LIN {X 0,Y 566.213,Z 135.454,A -85,B 0,C 180,E1 -2637.339,E2 -2637.339} C_VEL
LIN {X 0,Y 566.202,Z 135.458,A -85,B 0,C 180,E1 -2639.768,E2 -2639.768} C_VEL
LIN {X 0,Y 566.206,Z 135.453,A -85,B 0,C 180,E1 -2642.43,E2 -2642.43} C_VEL
LIN {X 0,Y 566.181,Z 135.454,A -85,B 0,C 180,E1 -2644.989,E2 -2644.989} C_VEL
LIN {X 0,Y 566.197,Z 135.457,A -85,B 0,C 180,E1 -2647.46,E2 -2647.46} C_VEL
LIN {X 0,Y 566.21,Z 135.449,A -85,B 0,C 180,E1 -2650.198,E2 -2650.198} C_VEL
LIN {X 0,Y 566.2,Z 135.453,A -85,B 0,C 180,E1 -2653.054,E2 -2653.054} C_VEL
LIN {X 0,Y 566.198,Z 135.454,A -85,B 0,C 180,E1 -2656.048,E2 -2656.048} C_VEL
LIN {X 0,Y 566.203,Z 135.457,A -85,B 0,C 180,E1 -2659.214,E2 -2659.214} C_VEL
LIN {X 0,Y 566.184,Z 135.459,A -85,B 0,C 180,E1 -2661.636,E2 -2661.636} C_VEL
LIN {X 0,Y 566.164,Z 135.455,A -85,B 0,C 180,E1 -2664.308,E2 -2664.308} C_VEL
LIN {X 0,Y 566.228,Z 135.449,A -85,B 0,C 180,E1 -2666.898,E2 -2666.898} C_VEL
LIN {X 0,Y 566.186,Z 135.459,A -85,B 0,C 180,E1 -2669.407,E2 -2669.407} C_VEL
LIN {X 0,Y 566.209,Z 135.448,A -85,B 0,C 180,E1 -2671.857,E2 -2671.857} C_VEL
LIN {X 0,Y 566.213,Z 135.447,A -85,B 0,C 180,E1 -2674.251,E2 -2674.251} C_VEL
LIN {X 0,Y 566.171,Z 135.46,A -85,B 0,C 180,E1 -2676.718,E2 -2676.718} C_VEL
LIN {X 0,Y 566.21,Z 135.448,A -85,B 0,C 180,E1 -2679.662,E2 -2679.662} C_VEL
LIN {X 0,Y 566.2,Z 135.454,A -85,B 0,C 180,E1 -2682.668,E2 -2682.668} C_VEL
LIN {X 0,Y 566.231,Z 135.447,A -85,B 0,C 180,E1 -2685.626,E2 -2685.626} C_VEL
LIN {X 0,Y 566.231,Z 135.453,A -85,B 0,C 180,E1 -2688.675,E2 -2688.675} C_VEL
LIN {X 0,Y 566.225,Z 135.445,A -85,B 0,C 180,E1 -2691.434,E2 -2691.434} C_VEL
LIN {X 0,Y 566.256,Z 135.45,A -85,B 0,C 180,E1 -2694.301,E2 -2694.301} C_VEL
LIN {X 0,Y 566.277,Z 135.442,A -85,B 0,C 180,E1 -2697.866,E2 -2697.866} C_VEL
LIN {X 0,Y 566.299,Z 135.44,A -85,B 0,C 180,E1 -2700.711,E2 -2700.711} C_VEL
LIN {X 0,Y 566.268,Z 135.444,A -85,B 0,C 180,E1 -2702.845,E2 -2702.845} C_VEL
LIN {X 0,Y 566.257,Z 135.446,A -85,B 0,C 180,E1 -2705.698,E2 -2705.698} C_VEL
LIN {X 0,Y 566.225,Z 135.448,A -85,B 0,C 180,E1 -2708.565,E2 -2708.565} C_VEL
LIN {X 0,Y 566.237,Z 135.445,A -85,B 0,C 180,E1 -2711.454,E2 -2711.454} C_VEL
LIN {X 0,Y 566.23,Z 135.45,A -85,B 0,C 180,E1 -2714.507,E2 -2714.507} C_VEL
LIN {X 0,Y 566.199,Z 135.452,A -85,B 0,C 180,E1 -2717.331,E2 -2717.331} C_VEL
LIN {X 0,Y 566.208,Z 135.451,A -85,B 0,C 180,E1 -2720.337,E2 -2720.337} C_VEL
LIN {X 0,Y 566.185,Z 135.457,A -85,B 0,C 180,E1 -2723.404,E2 -2723.404} C_VEL
LIN {X 0,Y 566.221,Z 135.455,A -85,B 0,C 180,E1 -2725.748,E2 -2725.748} C_VEL
LIN {X 0,Y 566.213,Z 135.45,A -85,B 0,C 180,E1 -2727.477,E2 -2727.477} C_VEL
LIN {X 0,Y 565.532,Z 135.536,A -85,B 0,C 180,E1 -2728.071,E2 -2728.071} C_VEL
LIN {X 0,Y 562.662,Z 135.892,A -85,B 0,C 180,E1 -2729.034,E2 -2729.034} C_VEL
LIN {X 0,Y 560.248,Z 136.199,A -85,B 0,C 180,E1 -2729.809,E2 -2729.809} C_VEL
LIN {X 0,Y 559.219,Z 136.322,A -85,B 0,C 180,E1 -2730.408,E2 -2730.408} C_VEL
LIN {X 0,Y 559.14,Z 136.331,A -85,B 0,C 180,E1 -2730.611,E2 -2730.611} C_VEL
LIN {X 0,Y 559.173,Z 136.331,A -85,B 0,C 180,E1 -2733.574,E2 -2733.574} C_VEL
LIN {X 0,Y 559.164,Z 136.328,A -85,B 0,C 180,E1 -2736.448,E2 -2736.448} C_VEL
LIN {X 0,Y 559.172,Z 136.33,A -85,B 0,C 180,E1 -2738.934,E2 -2738.934} C_VEL
LIN {X 0,Y 559.188,Z 136.327,A -85,B 0,C 180,E1 -2741.767,E2 -2741.767} C_VEL
LIN {X 0,Y 559.135,Z 136.334,A -85,B 0,C 180,E1 -2744.739,E2 -2744.739} C_VEL
LIN {X 0,Y 559.169,Z 136.319,A -85,B 0,C 180,E1 -2747.863,E2 -2747.863} C_VEL
LIN {X 0,Y 559.181,Z 136.324,A -85,B 0,C 180,E1 -2750.135,E2 -2750.135} C_VEL
LIN {X 0,Y 559.144,Z 136.339,A -85,B 0,C 180,E1 -2752.892,E2 -2752.892} C_VEL
LIN {X 0,Y 559.151,Z 136.327,A -85,B 0,C 180,E1 -2755.556,E2 -2755.556} C_VEL
LIN {X 0,Y 559.167,Z 136.329,A -85,B 0,C 180,E1 -2758.138,E2 -2758.138} C_VEL
LIN {X 0,Y 559.154,Z 136.334,A -85,B 0,C 180,E1 -2760.647,E2 -2760.647} C_VEL
LIN {X 0,Y 559.167,Z 136.331,A -85,B 0,C 180,E1 -2763.172,E2 -2763.172} C_VEL
LIN {X 0,Y 559.153,Z 136.33,A -85,B 0,C 180,E1 -2765.495,E2 -2765.495} C_VEL
LIN {X 0,Y 559.168,Z 136.337,A -85,B 0,C 180,E1 -2768.624,E2 -2768.624} C_VEL
LIN {X 0,Y 559.165,Z 136.332,A -85,B 0,C 180,E1 -2770.926,E2 -2770.926} C_VEL
LIN {X 0,Y 559.164,Z 136.332,A -85,B 0,C 180,E1 -2773.948,E2 -2773.948} C_VEL
LIN {X 0,Y 559.169,Z 136.335,A -85,B 0,C 180,E1 -2776.184,E2 -2776.184} C_VEL
LIN {X 0,Y 559.193,Z 136.326,A -85,B 0,C 180,E1 -2779.134,E2 -2779.134} C_VEL
LIN {X 0,Y 559.203,Z 136.332,A -85,B 0,C 180,E1 -2782.054,E2 -2782.054} C_VEL
LIN {X 0,Y 559.251,Z 136.319,A -85,B 0,C 180,E1 -2784.953,E2 -2784.953} C_VEL
LIN {X 0,Y 559.254,Z 136.324,A -85,B 0,C 180,E1 -2787.839,E2 -2787.839} C_VEL
LIN {X 0,Y 559.27,Z 136.317,A -85,B 0,C 180,E1 -2790.72,E2 -2790.72} C_VEL
LIN {X 0,Y 559.236,Z 136.32,A -85,B 0,C 180,E1 -2792.881,E2 -2792.881} C_VEL
LIN {X 0,Y 559.229,Z 136.329,A -85,B 0,C 180,E1 -2795.77,E2 -2795.77} C_VEL
LIN {X 0,Y 559.189,Z 136.326,A -85,B 0,C 180,E1 -2798.674,E2 -2798.674} C_VEL
LIN {X 0,Y 559.202,Z 136.332,A -85,B 0,C 180,E1 -2801.6,E2 -2801.6} C_VEL
LIN {X 0,Y 559.196,Z 136.325,A -85,B 0,C 180,E1 -2804.595,E2 -2804.595} C_VEL
LIN {X 0,Y 559.156,Z 136.338,A -85,B 0,C 180,E1 -2807.557,E2 -2807.557} C_VEL
LIN {X 0,Y 559.169,Z 136.332,A -85,B 0,C 180,E1 -2809.837,E2 -2809.837} C_VEL
LIN {X 0,Y 559.139,Z 136.333,A -85,B 0,C 180,E1 -2812.153,E2 -2812.153} C_VEL
LIN {X 0,Y 559.175,Z 136.334,A -85,B 0,C 180,E1 -2815.187,E2 -2815.187} C_VEL
LIN {X 0,Y 559.188,Z 136.328,A -85,B 0,C 180,E1 -2817.711,E2 -2817.711} C_VEL
LIN {X 0,Y 559.165,Z 136.327,A -85,B 0,C 180,E1 -2820.182,E2 -2820.182} C_VEL
LIN {X 0,Y 559.171,Z 136.331,A -85,B 0,C 180,E1 -2822.714,E2 -2822.714} C_VEL
LIN {X 0,Y 559.14,Z 136.335,A -85,B 0,C 180,E1 -2825.323,E2 -2825.323} C_VEL
LIN {X 0,Y 559.132,Z 136.332,A -85,B 0,C 180,E1 -2828.017,E2 -2828.017} C_VEL
LIN {X 0,Y 559.171,Z 136.331,A -85,B 0,C 180,E1 -2830.811,E2 -2830.811} C_VEL
LIN {X 0,Y 559.136,Z 136.328,A -85,B 0,C 180,E1 -2833.734,E2 -2833.734} C_VEL
LIN {X 0,Y 559.167,Z 136.337,A -85,B 0,C 180,E1 -2836.801,E2 -2836.801} C_VEL
LIN {X 0,Y 559.172,Z 136.327,A -85,B 0,C 180,E1 -2839.19,E2 -2839.19} C_VEL
LIN {X 0,Y 559.129,Z 136.334,A -85,B 0,C 180,E1 -2841.983,E2 -2841.983} C_VEL
LIN {X 0,Y 559.154,Z 136.331,A -85,B 0,C 180,E1 -2844.783,E2 -2844.783} C_VEL
LIN {X 0,Y 559.169,Z 136.327,A -85,B 0,C 180,E1 -2847.361,E2 -2847.361} C_VEL
LIN {X 0,Y 559.145,Z 136.336,A -85,B 0,C 180,E1 -2850.142,E2 -2850.142} C_VEL
LIN {X 0,Y 559.178,Z 136.323,A -85,B 0,C 180,E1 -2853.17,E2 -2853.17} C_VEL
LIN {X 0,Y 559.152,Z 136.329,A -85,B 0,C 180,E1 -2855.495,E2 -2855.495} C_VEL
LIN {X 0,Y 559.166,Z 136.329,A -85,B 0,C 180,E1 -2858.624,E2 -2858.624} C_VEL
LIN {X 0,Y 559.166,Z 136.322,A -85,B 0,C 180,E1 -2860.927,E2 -2860.927} C_VEL
LIN {X 0,Y 559.164,Z 136.335,A -85,B 0,C 180,E1 -2863.948,E2 -2863.948} C_VEL
LIN {X 0,Y 559.169,Z 136.333,A -85,B 0,C 180,E1 -2866.184,E2 -2866.184} C_VEL
LIN {X 0,Y 559.19,Z 136.321,A -85,B 0,C 180,E1 -2869.134,E2 -2869.134} C_VEL
LIN {X 0,Y 559.2,Z 136.328,A -85,B 0,C 180,E1 -2872.054,E2 -2872.054} C_VEL
LIN {X 0,Y 559.25,Z 136.318,A -85,B 0,C 180,E1 -2874.954,E2 -2874.954} C_VEL
LIN {X 0,Y 559.247,Z 136.321,A -85,B 0,C 180,E1 -2877.84,E2 -2877.84} C_VEL
LIN {X 0,Y 559.269,Z 136.31,A -85,B 0,C 180,E1 -2880.72,E2 -2880.72} C_VEL
LIN {X 0,Y 559.237,Z 136.319,A -85,B 0,C 180,E1 -2882.882,E2 -2882.882} C_VEL
LIN {X 0,Y 559.225,Z 136.324,A -85,B 0,C 180,E1 -2885.771,E2 -2885.771} C_VEL
LIN {X 0,Y 559.184,Z 136.322,A -85,B 0,C 180,E1 -2888.675,E2 -2888.675} C_VEL
LIN {X 0,Y 559.202,Z 136.327,A -85,B 0,C 180,E1 -2891.601,E2 -2891.601} C_VEL
LIN {X 0,Y 559.197,Z 136.325,A -85,B 0,C 180,E1 -2894.596,E2 -2894.596} C_VEL
LIN {X 0,Y 559.16,Z 136.327,A -85,B 0,C 180,E1 -2897.557,E2 -2897.557} C_VEL
LIN {X 0,Y 559.169,Z 136.325,A -85,B 0,C 180,E1 -2899.838,E2 -2899.838} C_VEL
LIN {X 0,Y 559.138,Z 136.331,A -85,B 0,C 180,E1 -2902.153,E2 -2902.153} C_VEL
LIN {X 0,Y 559.174,Z 136.328,A -85,B 0,C 180,E1 -2905.299,E2 -2905.299} C_VEL
LIN {X 0,Y 559.155,Z 136.326,A -85,B 0,C 180,E1 -2907.714,E2 -2907.714} C_VEL
LIN {X 0,Y 559.155,Z 136.33,A -85,B 0,C 180,E1 -2910.183,E2 -2910.183} C_VEL
LIN {X 0,Y 559.174,Z 136.334,A -85,B 0,C 180,E1 -2912.714,E2 -2912.714} C_VEL
LIN {X 0,Y 559.129,Z 136.333,A -85,B 0,C 180,E1 -2915.324,E2 -2915.324} C_VEL
LIN {X 0,Y 559.131,Z 136.334,A -85,B 0,C 180,E1 -2918.018,E2 -2918.018} C_VEL
LIN {X 0,Y 559.154,Z 136.334,A -85,B 0,C 180,E1 -2920.813,E2 -2920.813} C_VEL
LIN {X 0,Y 559.14,Z 136.331,A -85,B 0,C 180,E1 -2923.734,E2 -2923.734} C_VEL
LIN {X 0,Y 559.144,Z 136.334,A -85,B 0,C 180,E1 -2926.804,E2 -2926.804} C_VEL
LIN {X 0,Y 559.155,Z 136.325,A -85,B 0,C 180,E1 -2929.188,E2 -2929.188} C_VEL
LIN {X 0,Y 559.135,Z 136.337,A -85,B 0,C 180,E1 -2931.983,E2 -2931.983} C_VEL
LIN {X 0,Y 559.133,Z 136.333,A -85,B 0,C 180,E1 -2934.788,E2 -2934.788} C_VEL
LIN {X 0,Y 559.158,Z 136.329,A -85,B 0,C 180,E1 -2937.365,E2 -2937.365} C_VEL
LIN {X 0,Y 559.15,Z 136.337,A -85,B 0,C 180,E1 -2940.143,E2 -2940.143} C_VEL
LIN {X 0,Y 559.172,Z 136.331,A -85,B 0,C 180,E1 -2943.173,E2 -2943.173} C_VEL
LIN {X 0,Y 559.231,Z 136.477,A -85,B 0,C 180,E1 -2944.837,E2 -2944.837} C_VEL
LIN {X 0,Y 559.901,Z 140.893,A -85,B 0,C 180,E1 -2945.727,E2 -2945.727} C_VEL
LIN {X 0,Y 559.626,Z 156.438,A -85,B 0,C 180,E1 -2948.642,E2 -2948.642} C_VEL
LIN {X 0,Y 559.476,Z 170.036,A -85,B 0,C 180,E1 -2951.128,E2 -2951.128} C_VEL
LIN {X 0,Y 559.339,Z 184.658,A -85,B 0,C 180,E1 -2953.766,E2 -2953.766} C_VEL
LIN {X 0,Y 559.241,Z 196.165,A -85,B 0,C 180,E1 -2955.792,E2 -2955.792} C_VEL
LIN {X 0,Y 559.599,Z 198.54,A -85,B 0,C 180,E1 -2955.869,E2 -2955.869} C_VEL
LIN {X 0,Y 560.276,Z 204.023,A -85,B 0,C 180,E1 -2955.957,E2 -2955.957} C_VEL
LIN {X 0,Y 560.043,Z 301.149,A -85,B 0,C 180,E1 -2957.222,E2 -2957.222} C_VEL
LIN {X 0,Y 559.981,Z 311.04,A -85,B 0,C 180,E1 -2957.428,E2 -2957.428} C_VEL
LIN {X 0,Y 559.892,Z 321.006,A -85,B 0,C 180,E1 -2957.725,E2 -2957.725} C_VEL
LIN {X 0,Y 559.753,Z 330.356,A -85,B 0,C 180,E1 -2958.09,E2 -2958.09} C_VEL
LIN {X 0,Y 559.646,Z 339.669,A -85,B 0,C 180,E1 -2958.547,E2 -2958.547} C_VEL
LIN {X 0,Y 559.486,Z 349.449,A -85,B 0,C 180,E1 -2959.139,E2 -2959.139} C_VEL
LIN {X 0,Y 559.377,Z 358.154,A -85,B 0,C 180,E1 -2959.778,E2 -2959.778} C_VEL
LIN {X 0,Y 559.279,Z 365.525,A -85,B 0,C 180,E1 -2960.416,E2 -2960.416} C_VEL
LIN {X 0,Y 559.137,Z 372.717,A -85,B 0,C 180,E1 -2961.143,E2 -2961.143} C_VEL
LIN {X 0,Y 559.052,Z 380.264,A -85,B 0,C 180,E1 -2962.052,E2 -2962.052} C_VEL
LIN {X 0,Y 558.943,Z 386.554,A -85,B 0,C 180,E1 -2962.958,E2 -2962.958} C_VEL
LIN {X 0,Y 558.909,Z 391.787,A -85,B 0,C 180,E1 -2963.864,E2 -2963.864} C_VEL
LIN {X 0,Y 558.798,Z 396.885,A -85,B 0,C 180,E1 -2964.949,E2 -2964.949} C_VEL
LIN {X 0,Y 558.844,Z 400.843,A -85,B 0,C 180,E1 -2966.034,E2 -2966.034} C_VEL
LIN {X 0,Y 558.799,Z 403.767,A -85,B 0,C 180,E1 -2967.116,E2 -2967.116} C_VEL
LIN {X 0,Y 558.745,Z 406.194,A -85,B 0,C 180,E1 -2968.559,E2 -2968.559} C_VEL
LIN {X 0,Y 558.741,Z 406.778,A -85,B 0,C 180,E1 -2969.279,E2 -2969.279} C_VEL
LIN {X 0,Y 558.741,Z 406.778,A -85,B 0,C 180,E1 -2970.721,E2 -2970.721} C_VEL
LIN {X 0,Y 558.745,Z 406.194,A -85,B 0,C 180,E1 -2971.441,E2 -2971.441} C_VEL
LIN {X 0,Y 558.799,Z 403.767,A -85,B 0,C 180,E1 -2972.884,E2 -2972.884} C_VEL
LIN {X 0,Y 558.844,Z 400.843,A -85,B 0,C 180,E1 -2973.966,E2 -2973.966} C_VEL
LIN {X 0,Y 558.798,Z 396.885,A -85,B 0,C 180,E1 -2975.051,E2 -2975.051} C_VEL
LIN {X 0,Y 558.91,Z 391.787,A -85,B 0,C 180,E1 -2976.136,E2 -2976.136} C_VEL
LIN {X 0,Y 558.934,Z 386.668,A -85,B 0,C 180,E1 -2977.024,E2 -2977.024} C_VEL
LIN {X 0,Y 559.052,Z 380.264,A -85,B 0,C 180,E1 -2977.948,E2 -2977.948} C_VEL
LIN {X 0,Y 559.137,Z 372.717,A -85,B 0,C 180,E1 -2978.857,E2 -2978.857} C_VEL
LIN {X 0,Y 559.29,Z 363.612,A -85,B 0,C 180,E1 -2979.767,E2 -2979.767} C_VEL
LIN {X 0,Y 559.449,Z 352.147,A -85,B 0,C 180,E1 -2980.678,E2 -2980.678} C_VEL
LIN {X 0,Y 559.571,Z 343.177,A -85,B 0,C 180,E1 -2981.257,E2 -2981.257} C_VEL
LIN {X 0,Y 559.728,Z 333.771,A -85,B 0,C 180,E1 -2981.754,E2 -2981.754} C_VEL
LIN {X 0,Y 559.829,Z 323.581,A -85,B 0,C 180,E1 -2982.184,E2 -2982.184} C_VEL
LIN {X 0,Y 559.968,Z 313.661,A -85,B 0,C 180,E1 -2982.503,E2 -2982.503} C_VEL
LIN {X 0,Y 560.026,Z 303.813,A -85,B 0,C 180,E1 -2982.732,E2 -2982.732} C_VEL
LIN {X 0,Y 560.164,Z 279.204,A -85,B 0,C 180,E1 -2983.075,E2 -2983.075} C_VEL
LIN {X 0,Y 560.207,Z 202.231,A -85,B 0,C 180,E1 -2984.067,E2 -2984.067} C_VEL
LIN {X 0,Y 559.275,Z 196.499,A -85,B 0,C 180,E1 -2984.184,E2 -2984.184} C_VEL
LIN {X 0,Y 559.225,Z 195.089,A -85,B 0,C 180,E1 -2984.371,E2 -2984.371} C_VEL
LIN {X 0,Y 559.384,Z 178.831,A -85,B 0,C 180,E1 -2987.282,E2 -2987.282} C_VEL
LIN {X 0,Y 559.584,Z 162.717,A -85,B 0,C 180,E1 -2990.205,E2 -2990.205} C_VEL
LIN {X 0,Y 559.842,Z 146.337,A -85,B 0,C 180,E1 -2993.251,E2 -2993.251} C_VEL
LIN {X 0,Y 559.822,Z 139.871,A -85,B 0,C 180,E1 -2994.474,E2 -2994.474} C_VEL
LIN {X 0,Y 559.213,Z 136.373,A -85,B 0,C 180,E1 -2995.193,E2 -2995.193} C_VEL
LIN {X 0,Y 559.183,Z 136.333,A -85,B 0,C 180,E1 -2997.712,E2 -2997.712} C_VEL
LIN {X 0,Y 559.157,Z 136.337,A -85,B 0,C 180,E1 -3000.182,E2 -3000.182} C_VEL
LIN {X 0,Y 559.158,Z 136.329,A -85,B 0,C 180,E1 -3002.715,E2 -3002.715} C_VEL
LIN {X 0,Y 559.128,Z 136.334,A -85,B 0,C 180,E1 -3005.324,E2 -3005.324} C_VEL
LIN {X 0,Y 559.135,Z 136.337,A -85,B 0,C 180,E1 -3008.017,E2 -3008.017} C_VEL
LIN {X 0,Y 559.155,Z 136.325,A -85,B 0,C 180,E1 -3010.812,E2 -3010.812} C_VEL
LIN {X 0,Y 559.138,Z 136.338,A -85,B 0,C 180,E1 -3013.734,E2 -3013.734} C_VEL
LIN {X 0,Y 559.146,Z 136.331,A -85,B 0,C 180,E1 -3016.803,E2 -3016.803} C_VEL
LIN {X 0,Y 559.154,Z 136.334,A -85,B 0,C 180,E1 -3019.187,E2 -3019.187} C_VEL
LIN {X 0,Y 559.131,Z 136.334,A -85,B 0,C 180,E1 -3021.982,E2 -3021.982} C_VEL
LIN {X 0,Y 559.133,Z 136.333,A -85,B 0,C 180,E1 -3024.786,E2 -3024.786} C_VEL
LIN {X 0,Y 559.173,Z 136.334,A -85,B 0,C 180,E1 -3027.361,E2 -3027.361} C_VEL
LIN {X 0,Y 559.148,Z 136.33,A -85,B 0,C 180,E1 -3030.142,E2 -3030.142} C_VEL
LIN {X 0,Y 559.168,Z 136.332,A -85,B 0,C 180,E1 -3033.097,E2 -3033.097} C_VEL
LIN {X 0,Y 559.155,Z 136.331,A -85,B 0,C 180,E1 -3035.494,E2 -3035.494} C_VEL
LIN {X 0,Y 559.169,Z 136.331,A -85,B 0,C 180,E1 -3038.623,E2 -3038.623} C_VEL
LIN {X 0,Y 559.166,Z 136.331,A -85,B 0,C 180,E1 -3040.926,E2 -3040.926} C_VEL
LIN {X 0,Y 559.164,Z 136.327,A -85,B 0,C 180,E1 -3043.947,E2 -3043.947} C_VEL
LIN {X 0,Y 559.171,Z 136.328,A -85,B 0,C 180,E1 -3046.184,E2 -3046.184} C_VEL
LIN {X 0,Y 559.191,Z 136.322,A -85,B 0,C 180,E1 -3049.133,E2 -3049.133} C_VEL
LIN {X 0,Y 559.2,Z 136.322,A -85,B 0,C 180,E1 -3052.053,E2 -3052.053} C_VEL
LIN {X 0,Y 559.25,Z 136.32,A -85,B 0,C 180,E1 -3054.953,E2 -3054.953} C_VEL
LIN {X 0,Y 559.248,Z 136.318,A -85,B 0,C 180,E1 -3057.839,E2 -3057.839} C_VEL
LIN {X 0,Y 559.269,Z 136.315,A -85,B 0,C 180,E1 -3060.72,E2 -3060.72} C_VEL
LIN {X 0,Y 559.235,Z 136.32,A -85,B 0,C 180,E1 -3062.881,E2 -3062.881} C_VEL
LIN {X 0,Y 559.225,Z 136.323,A -85,B 0,C 180,E1 -3065.77,E2 -3065.77} C_VEL
LIN {X 0,Y 559.184,Z 136.323,A -85,B 0,C 180,E1 -3068.674,E2 -3068.674} C_VEL
LIN {X 0,Y 559.201,Z 136.322,A -85,B 0,C 180,E1 -3071.6,E2 -3071.6} C_VEL
LIN {X 0,Y 559.195,Z 136.326,A -85,B 0,C 180,E1 -3074.595,E2 -3074.595} C_VEL
LIN {X 0,Y 559.159,Z 136.331,A -85,B 0,C 180,E1 -3077.556,E2 -3077.556} C_VEL
LIN {X 0,Y 559.167,Z 136.331,A -85,B 0,C 180,E1 -3079.837,E2 -3079.837} C_VEL
LIN {X 0,Y 559.137,Z 136.335,A -85,B 0,C 180,E1 -3082.153,E2 -3082.153} C_VEL
LIN {X 0,Y 559.175,Z 136.328,A -85,B 0,C 180,E1 -3085.187,E2 -3085.187} C_VEL
LIN {X 0,Y 559.19,Z 136.33,A -85,B 0,C 180,E1 -3087.711,E2 -3087.711} C_VEL
LIN {X 0,Y 559.14,Z 136.331,A -85,B 0,C 180,E1 -3090.611,E2 -3090.611} C_VEL
LIN {X 0,Y 558.481,Z 136.419,A -85,B 0,C 180,E1 -3091.212,E2 -3091.212} C_VEL
LIN {X 0,Y 555.622,Z 136.771,A -85,B 0,C 180,E1 -3092.188,E2 -3092.188} C_VEL
LIN {X 0,Y 553.211,Z 137.071,A -85,B 0,C 180,E1 -3092.974,E2 -3092.974} C_VEL
LIN {X 0,Y 552.192,Z 137.2,A -85,B 0,C 180,E1 -3093.581,E2 -3093.581} C_VEL
LIN {X 0,Y 552.118,Z 137.203,A -85,B 0,C 180,E1 -3093.786,E2 -3093.786} C_VEL
LIN {X 0,Y 552.107,Z 137.208,A -85,B 0,C 180,E1 -3096.746,E2 -3096.746} C_VEL
LIN {X 0,Y 552.129,Z 137.208,A -85,B 0,C 180,E1 -3099.527,E2 -3099.527} C_VEL
LIN {X 0,Y 552.126,Z 137.205,A -85,B 0,C 180,E1 -3102.425,E2 -3102.425} C_VEL
LIN {X 0,Y 552.092,Z 137.209,A -85,B 0,C 180,E1 -3105.563,E2 -3105.563} C_VEL
LIN {X 0,Y 552.134,Z 137.198,A -85,B 0,C 180,E1 -3108.676,E2 -3108.676} C_VEL
LIN {X 0,Y 552.116,Z 137.21,A -85,B 0,C 180,E1 -3111.411,E2 -3111.411} C_VEL
LIN {X 0,Y 552.109,Z 137.205,A -85,B 0,C 180,E1 -3114.159,E2 -3114.159} C_VEL
LIN {X 0,Y 552.119,Z 137.21,A -85,B 0,C 180,E1 -3116.815,E2 -3116.815} C_VEL
LIN {X 0,Y 552.11,Z 137.207,A -85,B 0,C 180,E1 -3119.392,E2 -3119.392} C_VEL
LIN {X 0,Y 552.119,Z 137.205,A -85,B 0,C 180,E1 -3121.903,E2 -3121.903} C_VEL
LIN {X 0,Y 552.152,Z 137.211,A -85,B 0,C 180,E1 -3124.65,E2 -3124.65} C_VEL
LIN {X 0,Y 552.093,Z 137.21,A -85,B 0,C 180,E1 -3127.549,E2 -3127.549} C_VEL
LIN {X 0,Y 552.153,Z 137.209,A -85,B 0,C 180,E1 -3130.675,E2 -3130.675} C_VEL
LIN {X 0,Y 552.114,Z 137.208,A -85,B 0,C 180,E1 -3133.737,E2 -3133.737} C_VEL
LIN {X 0,Y 552.133,Z 137.209,A -85,B 0,C 180,E1 -3136.005,E2 -3136.005} C_VEL
LIN {X 0,Y 552.16,Z 137.203,A -85,B 0,C 180,E1 -3138.993,E2 -3138.993} C_VEL
LIN {X 0,Y 552.157,Z 137.208,A -85,B 0,C 180,E1 -3141.952,E2 -3141.952} C_VEL
LIN {X 0,Y 552.226,Z 137.194,A -85,B 0,C 180,E1 -3144.889,E2 -3144.889} C_VEL
LIN {X 0,Y 552.225,Z 137.2,A -85,B 0,C 180,E1 -3147.812,E2 -3147.812} C_VEL
LIN {X 0,Y 552.24,Z 137.193,A -85,B 0,C 180,E1 -3150.729,E2 -3150.729} C_VEL
LIN {X 0,Y 552.203,Z 137.197,A -85,B 0,C 180,E1 -3152.918,E2 -3152.918} C_VEL
LIN {X 0,Y 552.199,Z 137.205,A -85,B 0,C 180,E1 -3155.844,E2 -3155.844} C_VEL
LIN {X 0,Y 552.16,Z 137.202,A -85,B 0,C 180,E1 -3158.786,E2 -3158.786} C_VEL
LIN {X 0,Y 552.16,Z 137.21,A -85,B 0,C 180,E1 -3161.75,E2 -3161.75} C_VEL
LIN {X 0,Y 552.133,Z 137.205,A -85,B 0,C 180,E1 -3164.748,E2 -3164.748} C_VEL
LIN {X 0,Y 552.108,Z 137.214,A -85,B 0,C 180,E1 -3167.788,E2 -3167.788} C_VEL
LIN {X 0,Y 552.128,Z 137.207,A -85,B 0,C 180,E1 -3170.101,E2 -3170.101} C_VEL
LIN {X 0,Y 552.093,Z 137.21,A -85,B 0,C 180,E1 -3172.451,E2 -3172.451} C_VEL
LIN {X 0,Y 552.152,Z 137.211,A -85,B 0,C 180,E1 -3175.35,E2 -3175.35} C_VEL
LIN {X 0,Y 552.121,Z 137.205,A -85,B 0,C 180,E1 -3178.097,E2 -3178.097} C_VEL
LIN {X 0,Y 552.11,Z 137.207,A -85,B 0,C 180,E1 -3180.608,E2 -3180.608} C_VEL
LIN {X 0,Y 552.118,Z 137.21,A -85,B 0,C 180,E1 -3183.185,E2 -3183.185} C_VEL
LIN {X 0,Y 552.099,Z 137.207,A -85,B 0,C 180,E1 -3185.842,E2 -3185.842} C_VEL
LIN {X 0,Y 552.122,Z 137.211,A -85,B 0,C 180,E1 -3189.062,E2 -3189.062} C_VEL
LIN {X 0,Y 552.133,Z 137.196,A -85,B 0,C 180,E1 -3191.444,E2 -3191.444} C_VEL
LIN {X 0,Y 552.09,Z 137.21,A -85,B 0,C 180,E1 -3194.532,E2 -3194.532} C_VEL
LIN {X 0,Y 552.126,Z 137.204,A -85,B 0,C 180,E1 -3197.584,E2 -3197.584} C_VEL
LIN {X 0,Y 552.129,Z 137.208,A -85,B 0,C 180,E1 -3200.473,E2 -3200.473} C_VEL
LIN {X 0,Y 552.11,Z 137.207,A -85,B 0,C 180,E1 -3203.316,E2 -3203.316} C_VEL
LIN {X 0,Y 552.135,Z 137.201,A -85,B 0,C 180,E1 -3205.94,E2 -3205.94} C_VEL
LIN {X 0,Y 552.113,Z 137.215,A -85,B 0,C 180,E1 -3208.541,E2 -3208.541} C_VEL
LIN {X 0,Y 552.121,Z 137.203,A -85,B 0,C 180,E1 -3211.438,E2 -3211.438} C_VEL
LIN {X 0,Y 552.133,Z 137.211,A -85,B 0,C 180,E1 -3214.356,E2 -3214.356} C_VEL
LIN {X 0,Y 552.105,Z 137.209,A -85,B 0,C 180,E1 -3216.759,E2 -3216.759} C_VEL
LIN {X 0,Y 552.115,Z 137.204,A -85,B 0,C 180,E1 -3219.12,E2 -3219.12} C_VEL
LIN {X 0,Y 552.126,Z 137.2,A -85,B 0,C 180,E1 -3221.445,E2 -3221.445} C_VEL
LIN {X 0,Y 552.113,Z 137.209,A -85,B 0,C 180,E1 -3223.738,E2 -3223.738} C_VEL
LIN {X 0,Y 552.132,Z 137.213,A -85,B 0,C 180,E1 -3226.005,E2 -3226.005} C_VEL
LIN {X 0,Y 552.157,Z 137.197,A -85,B 0,C 180,E1 -3228.994,E2 -3228.994} C_VEL
LIN {X 0,Y 552.154,Z 137.207,A -85,B 0,C 180,E1 -3231.952,E2 -3231.952} C_VEL
LIN {X 0,Y 552.225,Z 137.192,A -85,B 0,C 180,E1 -3234.889,E2 -3234.889} C_VEL
LIN {X 0,Y 552.219,Z 137.196,A -85,B 0,C 180,E1 -3237.812,E2 -3237.812} C_VEL
LIN {X 0,Y 552.239,Z 137.185,A -85,B 0,C 180,E1 -3240.73,E2 -3240.73} C_VEL
LIN {X 0,Y 552.203,Z 137.195,A -85,B 0,C 180,E1 -3242.919,E2 -3242.919} C_VEL
LIN {X 0,Y 552.196,Z 137.199,A -85,B 0,C 180,E1 -3245.844,E2 -3245.844} C_VEL
LIN {X 0,Y 552.155,Z 137.198,A -85,B 0,C 180,E1 -3248.786,E2 -3248.786} C_VEL
LIN {X 0,Y 552.16,Z 137.202,A -85,B 0,C 180,E1 -3251.751,E2 -3251.751} C_VEL
LIN {X 0,Y 552.134,Z 137.206,A -85,B 0,C 180,E1 -3254.749,E2 -3254.749} C_VEL
LIN {X 0,Y 552.11,Z 137.202,A -85,B 0,C 180,E1 -3257.789,E2 -3257.789} C_VEL
LIN {X 0,Y 552.128,Z 137.201,A -85,B 0,C 180,E1 -3260.102,E2 -3260.102} C_VEL
LIN {X 0,Y 552.09,Z 137.21,A -85,B 0,C 180,E1 -3262.451,E2 -3262.451} C_VEL
LIN {X 0,Y 552.154,Z 137.201,A -85,B 0,C 180,E1 -3265.351,E2 -3265.351} C_VEL
LIN {X 0,Y 552.107,Z 137.204,A -85,B 0,C 180,E1 -3268.099,E2 -3268.099} C_VEL
LIN {X 0,Y 552.106,Z 137.213,A -85,B 0,C 180,E1 -3270.609,E2 -3270.609} C_VEL
LIN {X 0,Y 552.122,Z 137.205,A -85,B 0,C 180,E1 -3273.186,E2 -3273.186} C_VEL
LIN {X 0,Y 552.086,Z 137.209,A -85,B 0,C 180,E1 -3275.844,E2 -3275.844} C_VEL
LIN {X 0,Y 552.12,Z 137.206,A -85,B 0,C 180,E1 -3279.062,E2 -3279.062} C_VEL
LIN {X 0,Y 552.12,Z 137.205,A -85,B 0,C 180,E1 -3281.446,E2 -3281.446} C_VEL
LIN {X 0,Y 552.093,Z 137.216,A -85,B 0,C 180,E1 -3284.532,E2 -3284.532} C_VEL
LIN {X 0,Y 552.129,Z 137.205,A -85,B 0,C 180,E1 -3287.585,E2 -3287.585} C_VEL
LIN {X 0,Y 552.134,Z 137.21,A -85,B 0,C 180,E1 -3290.474,E2 -3290.474} C_VEL
LIN {X 0,Y 552.107,Z 137.207,A -85,B 0,C 180,E1 -3293.317,E2 -3293.317} C_VEL
LIN {X 0,Y 552.128,Z 137.21,A -85,B 0,C 180,E1 -3295.94,E2 -3295.94} C_VEL
LIN {X 0,Y 552.121,Z 137.21,A -85,B 0,C 180,E1 -3298.541,E2 -3298.541} C_VEL
LIN {X 0,Y 552.106,Z 137.211,A -85,B 0,C 180,E1 -3301.442,E2 -3301.442} C_VEL
LIN {X 0,Y 552.135,Z 137.213,A -85,B 0,C 180,E1 -3304.356,E2 -3304.356} C_VEL
LIN {X 0,Y 552.163,Z 137.377,A -85,B 0,C 180,E1 -3304.684,E2 -3304.684} C_VEL
LIN {X 0,Y 552.952,Z 142.881,A -85,B 0,C 180,E1 -3305.802,E2 -3305.802} C_VEL
LIN {X 0,Y 552.651,Z 160.492,A -85,B 0,C 180,E1 -3309.141,E2 -3309.141} C_VEL
LIN {X 0,Y 552.461,Z 176.175,A -85,B 0,C 180,E1 -3312.032,E2 -3312.032} C_VEL
LIN {X 0,Y 552.221,Z 193.889,A -85,B 0,C 180,E1 -3315.254,E2 -3315.254} C_VEL
LIN {X 0,Y 552.194,Z 196.156,A -85,B 0,C 180,E1 -3315.621,E2 -3315.621} C_VEL
LIN {X 0,Y 553.383,Z 204.134,A -85,B 0,C 180,E1 -3315.783,E2 -3315.783} C_VEL
LIN {X 0,Y 553.136,Z 300.958,A -85,B 0,C 180,E1 -3317.06,E2 -3317.06} C_VEL
LIN {X 0,Y 553.044,Z 310.855,A -85,B 0,C 180,E1 -3317.268,E2 -3317.268} C_VEL
LIN {X 0,Y 552.962,Z 320.834,A -85,B 0,C 180,E1 -3317.569,E2 -3317.569} C_VEL
LIN {X 0,Y 552.765,Z 331.199,A -85,B 0,C 180,E1 -3317.983,E2 -3317.983} C_VEL
LIN {X 0,Y 552.64,Z 340.439,A -85,B 0,C 180,E1 -3318.452,E2 -3318.452} C_VEL
LIN {X 0,Y 552.496,Z 349.338,A -85,B 0,C 180,E1 -3319,E2 -3319} C_VEL
LIN {X 0,Y 552.383,Z 358.071,A -85,B 0,C 180,E1 -3319.647,E2 -3319.647} C_VEL
LIN {X 0,Y 552.243,Z 365.468,A -85,B 0,C 180,E1 -3320.292,E2 -3320.292} C_VEL
LIN {X 0,Y 552.099,Z 372.688,A -85,B 0,C 180,E1 -3321.029,E2 -3321.029} C_VEL
LIN {X 0,Y 552.01,Z 378.884,A -85,B 0,C 180,E1 -3321.765,E2 -3321.765} C_VEL
LIN {X 0,Y 551.904,Z 385.392,A -85,B 0,C 180,E1 -3322.684,E2 -3322.684} C_VEL
LIN {X 0,Y 551.808,Z 391.081,A -85,B 0,C 180,E1 -3323.651,E2 -3323.651} C_VEL
LIN {X 0,Y 551.802,Z 395.331,A -85,B 0,C 180,E1 -3324.519,E2 -3324.519} C_VEL
LIN {X 0,Y 551.766,Z 399.626,A -85,B 0,C 180,E1 -3325.617,E2 -3325.617} C_VEL
LIN {X 0,Y 551.75,Z 401.973,A -85,B 0,C 180,E1 -3326.349,E2 -3326.349} C_VEL
LIN {X 0,Y 551.723,Z 403.76,A -85,B 0,C 180,E1 -3327.079,E2 -3327.079} C_VEL
LIN {X 0,Y 551.645,Z 406.185,A -85,B 0,C 180,E1 -3328.54,E2 -3328.54} C_VEL
LIN {X 0,Y 551.641,Z 406.769,A -85,B 0,C 180,E1 -3329.27,E2 -3329.27} C_VEL
LIN {X 0,Y 551.641,Z 406.769,A -85,B 0,C 180,E1 -3330.73,E2 -3330.73} C_VEL
LIN {X 0,Y 551.645,Z 406.185,A -85,B 0,C 180,E1 -3331.46,E2 -3331.46} C_VEL
LIN {X 0,Y 551.723,Z 403.76,A -85,B 0,C 180,E1 -3332.921,E2 -3332.921} C_VEL
LIN {X 0,Y 551.764,Z 400.835,A -85,B 0,C 180,E1 -3334.017,E2 -3334.017} C_VEL
LIN {X 0,Y 551.723,Z 396.875,A -85,B 0,C 180,E1 -3335.116,E2 -3335.116} C_VEL
LIN {X 0,Y 551.837,Z 392.381,A -85,B 0,C 180,E1 -3336.098,E2 -3336.098} C_VEL
LIN {X 0,Y 551.886,Z 386.542,A -85,B 0,C 180,E1 -3337.132,E2 -3337.132} C_VEL
LIN {X 0,Y 551.984,Z 380.254,A -85,B 0,C 180,E1 -3338.051,E2 -3338.051} C_VEL
LIN {X 0,Y 552.071,Z 374.315,A -85,B 0,C 180,E1 -3338.787,E2 -3338.787} C_VEL
LIN {X 0,Y 552.199,Z 367.387,A -85,B 0,C 180,E1 -3339.524,E2 -3339.524} C_VEL
LIN {X 0,Y 552.339,Z 359.205,A -85,B 0,C 180,E1 -3340.261,E2 -3340.261} C_VEL
LIN {X 0,Y 552.462,Z 350.69,A -85,B 0,C 180,E1 -3340.908,E2 -3340.908} C_VEL
LIN {X 0,Y 552.621,Z 341.516,A -85,B 0,C 180,E1 -3341.487,E2 -3341.487} C_VEL
LIN {X 0,Y 552.789,Z 332.208,A -85,B 0,C 180,E1 -3341.969,E2 -3341.969} C_VEL
LIN {X 0,Y 552.88,Z 323.409,A -85,B 0,C 180,E1 -3342.34,E2 -3342.34} C_VEL
LIN {X 0,Y 553.031,Z 313.479,A -85,B 0,C 180,E1 -3342.663,E2 -3342.663} C_VEL
LIN {X 0,Y 553.096,Z 303.621,A -85,B 0,C 180,E1 -3342.895,E2 -3342.895} C_VEL
LIN {X 0,Y 553.264,Z 279.013,A -85,B 0,C 180,E1 -3343.241,E2 -3343.241} C_VEL
LIN {X 0,Y 553.295,Z 202.739,A -85,B 0,C 180,E1 -3344.238,E2 -3344.238} C_VEL
LIN {X 0,Y 552.213,Z 196.154,A -85,B 0,C 180,E1 -3344.379,E2 -3344.379} C_VEL
LIN {X 0,Y 552.334,Z 181.396,A -85,B 0,C 180,E1 -3347.017,E2 -3347.017} C_VEL
LIN {X 0,Y 552.558,Z 166.516,A -85,B 0,C 180,E1 -3349.744,E2 -3349.744} C_VEL
LIN {X 0,Y 552.778,Z 151.217,A -85,B 0,C 180,E1 -3352.618,E2 -3352.618} C_VEL
LIN {X 0,Y 552.92,Z 141.865,A -85,B 0,C 180,E1 -3354.399,E2 -3354.399} C_VEL
LIN {X 0,Y 552.162,Z 137.233,A -85,B 0,C 180,E1 -3355.363,E2 -3355.363} C_VEL
LIN {X 0,Y 552.108,Z 137.215,A -85,B 0,C 180,E1 -3358.098,E2 -3358.098} C_VEL
LIN {X 0,Y 552.108,Z 137.21,A -85,B 0,C 180,E1 -3360.609,E2 -3360.609} C_VEL
LIN {X 0,Y 552.117,Z 137.207,A -85,B 0,C 180,E1 -3363.185,E2 -3363.185} C_VEL
LIN {X 0,Y 552.086,Z 137.215,A -85,B 0,C 180,E1 -3365.843,E2 -3365.843} C_VEL
LIN {X 0,Y 552.126,Z 137.205,A -85,B 0,C 180,E1 -3369.061,E2 -3369.061} C_VEL
LIN {X 0,Y 552.12,Z 137.207,A -85,B 0,C 180,E1 -3371.445,E2 -3371.445} C_VEL
LIN {X 0,Y 552.09,Z 137.209,A -85,B 0,C 180,E1 -3374.531,E2 -3374.531} C_VEL
LIN {X 0,Y 552.129,Z 137.213,A -85,B 0,C 180,E1 -3377.584,E2 -3377.584} C_VEL
LIN {X 0,Y 552.128,Z 137.202,A -85,B 0,C 180,E1 -3380.472,E2 -3380.472} C_VEL
LIN {X 0,Y 552.105,Z 137.217,A -85,B 0,C 180,E1 -3383.316,E2 -3383.316} C_VEL
LIN {X 0,Y 552.128,Z 137.202,A -85,B 0,C 180,E1 -3385.939,E2 -3385.939} C_VEL
LIN {X 0,Y 552.117,Z 137.206,A -85,B 0,C 180,E1 -3388.54,E2 -3388.54} C_VEL
LIN {X 0,Y 552.123,Z 137.207,A -85,B 0,C 180,E1 -3391.437,E2 -3391.437} C_VEL
LIN {X 0,Y 552.129,Z 137.202,A -85,B 0,C 180,E1 -3394.355,E2 -3394.355} C_VEL
LIN {X 0,Y 552.097,Z 137.213,A -85,B 0,C 180,E1 -3396.757,E2 -3396.757} C_VEL
LIN {X 0,Y 552.118,Z 137.209,A -85,B 0,C 180,E1 -3399.119,E2 -3399.119} C_VEL
LIN {X 0,Y 552.125,Z 137.201,A -85,B 0,C 180,E1 -3401.444,E2 -3401.444} C_VEL
LIN {X 0,Y 552.114,Z 137.204,A -85,B 0,C 180,E1 -3403.737,E2 -3403.737} C_VEL
LIN {X 0,Y 552.134,Z 137.204,A -85,B 0,C 180,E1 -3406.004,E2 -3406.004} C_VEL
LIN {X 0,Y 552.158,Z 137.199,A -85,B 0,C 180,E1 -3408.993,E2 -3408.993} C_VEL
LIN {X 0,Y 552.154,Z 137.198,A -85,B 0,C 180,E1 -3411.951,E2 -3411.951} C_VEL
LIN {X 0,Y 552.225,Z 137.196,A -85,B 0,C 180,E1 -3414.889,E2 -3414.889} C_VEL
LIN {X 0,Y 552.22,Z 137.193,A -85,B 0,C 180,E1 -3417.811,E2 -3417.811} C_VEL
LIN {X 0,Y 552.239,Z 137.19,A -85,B 0,C 180,E1 -3420.729,E2 -3420.729} C_VEL
LIN {X 0,Y 552.202,Z 137.196,A -85,B 0,C 180,E1 -3422.918,E2 -3422.918} C_VEL
LIN {X 0,Y 552.196,Z 137.2,A -85,B 0,C 180,E1 -3425.844,E2 -3425.844} C_VEL
LIN {X 0,Y 552.155,Z 137.197,A -85,B 0,C 180,E1 -3428.785,E2 -3428.785} C_VEL
LIN {X 0,Y 552.158,Z 137.201,A -85,B 0,C 180,E1 -3431.75,E2 -3431.75} C_VEL
LIN {X 0,Y 552.132,Z 137.204,A -85,B 0,C 180,E1 -3434.748,E2 -3434.748} C_VEL
LIN {X 0,Y 552.11,Z 137.212,A -85,B 0,C 180,E1 -3437.788,E2 -3437.788} C_VEL
LIN {X 0,Y 552.126,Z 137.208,A -85,B 0,C 180,E1 -3440.101,E2 -3440.101} C_VEL
LIN {X 0,Y 552.091,Z 137.21,A -85,B 0,C 180,E1 -3442.451,E2 -3442.451} C_VEL
LIN {X 0,Y 552.152,Z 137.205,A -85,B 0,C 180,E1 -3445.351,E2 -3445.351} C_VEL
LIN {X 0,Y 552.121,Z 137.206,A -85,B 0,C 180,E1 -3448.097,E2 -3448.097} C_VEL
LIN {X 0,Y 552.102,Z 137.208,A -85,B 0,C 180,E1 -3450.609,E2 -3450.609} C_VEL
LIN {X 0,Y 552.124,Z 137.209,A -85,B 0,C 180,E1 -3453.185,E2 -3453.185} C_VEL
LIN {X 0,Y 552.118,Z 137.203,A -85,B 0,C 180,E1 -3453.786,E2 -3453.786} C_VEL
LIN {X 0,Y 551.482,Z 137.284,A -85,B 0,C 180,E1 -3454.395,E2 -3454.395} C_VEL
LIN {X 0,Y 548.658,Z 137.641,A -85,B 0,C 180,E1 -3455.383,E2 -3455.383} C_VEL
LIN {X 0,Y 546.234,Z 137.94,A -85,B 0,C 180,E1 -3456.178,E2 -3456.178} C_VEL
LIN {X 0,Y 545.164,Z 138.073,A -85,B 0,C 180,E1 -3456.792,E2 -3456.792} C_VEL
LIN {X 0,Y 545.061,Z 138.088,A -85,B 0,C 180,E1 -3457,E2 -3457} C_VEL
LIN {X 0,Y 545.069,Z 138.081,A -85,B 0,C 180,E1 -3460.142,E2 -3460.142} C_VEL
LIN {X 0,Y 545.083,Z 138.089,A -85,B 0,C 180,E1 -3463.105,E2 -3463.105} C_VEL
LIN {X 0,Y 545.062,Z 138.08,A -85,B 0,C 180,E1 -3466.224,E2 -3466.224} C_VEL
LIN {X 0,Y 545.091,Z 138.077,A -85,B 0,C 180,E1 -3468.887,E2 -3468.887} C_VEL
LIN {X 0,Y 545.05,Z 138.087,A -85,B 0,C 180,E1 -3471.763,E2 -3471.763} C_VEL
LIN {X 0,Y 545.06,Z 138.086,A -85,B 0,C 180,E1 -3474.534,E2 -3474.534} C_VEL
LIN {X 0,Y 545.077,Z 138.088,A -85,B 0,C 180,E1 -3477.213,E2 -3477.213} C_VEL
LIN {X 0,Y 545.098,Z 138.079,A -85,B 0,C 180,E1 -3479.813,E2 -3479.813} C_VEL
LIN {X 0,Y 545.091,Z 138.09,A -85,B 0,C 180,E1 -3482.826,E2 -3482.826} C_VEL
LIN {X 0,Y 545.048,Z 138.087,A -85,B 0,C 180,E1 -3485.631,E2 -3485.631} C_VEL
LIN {X 0,Y 545.063,Z 138.091,A -85,B 0,C 180,E1 -3488.837,E2 -3488.837} C_VEL
LIN {X 0,Y 545.077,Z 138.085,A -85,B 0,C 180,E1 -3491.196,E2 -3491.196} C_VEL
LIN {X 0,Y 545.07,Z 138.085,A -85,B 0,C 180,E1 -3493.521,E2 -3493.521} C_VEL
LIN {X 0,Y 545.092,Z 138.084,A -85,B 0,C 180,E1 -3495.82,E2 -3495.82} C_VEL
LIN {X 0,Y 545.116,Z 138.082,A -85,B 0,C 180,E1 -3498.849,E2 -3498.849} C_VEL
LIN {X 0,Y 545.127,Z 138.082,A -85,B 0,C 180,E1 -3501.847,E2 -3501.847} C_VEL
LIN {X 0,Y 545.202,Z 138.07,A -85,B 0,C 180,E1 -3504.823,E2 -3504.823} C_VEL
LIN {X 0,Y 545.196,Z 138.075,A -85,B 0,C 180,E1 -3507.784,E2 -3507.784} C_VEL
LIN {X 0,Y 545.21,Z 138.069,A -85,B 0,C 180,E1 -3510.739,E2 -3510.739} C_VEL
LIN {X 0,Y 545.169,Z 138.073,A -85,B 0,C 180,E1 -3512.956,E2 -3512.956} C_VEL
LIN {X 0,Y 545.171,Z 138.08,A -85,B 0,C 180,E1 -3515.919,E2 -3515.919} C_VEL
LIN {X 0,Y 545.118,Z 138.08,A -85,B 0,C 180,E1 -3518.9,E2 -3518.9} C_VEL
LIN {X 0,Y 545.132,Z 138.083,A -85,B 0,C 180,E1 -3521.904,E2 -3521.904} C_VEL
LIN {X 0,Y 545.082,Z 138.085,A -85,B 0,C 180,E1 -3524.944,E2 -3524.944} C_VEL
LIN {X 0,Y 545.076,Z 138.087,A -85,B 0,C 180,E1 -3528.026,E2 -3528.026} C_VEL
LIN {X 0,Y 545.092,Z 138.082,A -85,B 0,C 180,E1 -3530.372,E2 -3530.372} C_VEL
LIN {X 0,Y 545.088,Z 138.089,A -85,B 0,C 180,E1 -3533.559,E2 -3533.559} C_VEL
LIN {X 0,Y 545.076,Z 138.085,A -85,B 0,C 180,E1 -3536,E2 -3536} C_VEL
LIN {X 0,Y 545.088,Z 138.083,A -85,B 0,C 180,E1 -3538.749,E2 -3538.749} C_VEL
LIN {X 0,Y 545.074,Z 138.086,A -85,B 0,C 180,E1 -3541.682,E2 -3541.682} C_VEL
LIN {X 0,Y 545.072,Z 138.081,A -85,B 0,C 180,E1 -3544.563,E2 -3544.563} C_VEL
LIN {X 0,Y 545.035,Z 138.094,A -85,B 0,C 180,E1 -3547.304,E2 -3547.304} C_VEL
LIN {X 0,Y 545.07,Z 138.082,A -85,B 0,C 180,E1 -3550.142,E2 -3550.142} C_VEL
LIN {X 0,Y 545.073,Z 138.085,A -85,B 0,C 180,E1 -3553.107,E2 -3553.107} C_VEL
LIN {X 0,Y 545.061,Z 138.087,A -85,B 0,C 180,E1 -3556.224,E2 -3556.224} C_VEL
LIN {X 0,Y 545.092,Z 138.085,A -85,B 0,C 180,E1 -3558.887,E2 -3558.887} C_VEL
LIN {X 0,Y 545.048,Z 138.087,A -85,B 0,C 180,E1 -3561.763,E2 -3561.763} C_VEL
LIN {X 0,Y 545.06,Z 138.09,A -85,B 0,C 180,E1 -3564.534,E2 -3564.534} C_VEL
LIN {X 0,Y 545.078,Z 138.083,A -85,B 0,C 180,E1 -3567.213,E2 -3567.213} C_VEL
LIN {X 0,Y 545.061,Z 138.087,A -85,B 0,C 180,E1 -3569.811,E2 -3569.811} C_VEL
LIN {X 0,Y 545.091,Z 138.084,A -85,B 0,C 180,E1 -3572.345,E2 -3572.345} C_VEL
LIN {X 0,Y 545.113,Z 138.08,A -85,B 0,C 180,E1 -3574.821,E2 -3574.821} C_VEL
LIN {X 0,Y 545.039,Z 138.087,A -85,B 0,C 180,E1 -3577.243,E2 -3577.243} C_VEL
LIN {X 0,Y 545.115,Z 138.076,A -85,B 0,C 180,E1 -3580.415,E2 -3580.415} C_VEL
LIN {X 0,Y 545.069,Z 138.084,A -85,B 0,C 180,E1 -3583.522,E2 -3583.522} C_VEL
LIN {X 0,Y 545.091,Z 138.088,A -85,B 0,C 180,E1 -3585.82,E2 -3585.82} C_VEL
LIN {X 0,Y 545.113,Z 138.074,A -85,B 0,C 180,E1 -3588.85,E2 -3588.85} C_VEL
LIN {X 0,Y 545.125,Z 138.081,A -85,B 0,C 180,E1 -3591.847,E2 -3591.847} C_VEL
LIN {X 0,Y 545.201,Z 138.067,A -85,B 0,C 180,E1 -3594.823,E2 -3594.823} C_VEL
LIN {X 0,Y 545.191,Z 138.071,A -85,B 0,C 180,E1 -3597.784,E2 -3597.784} C_VEL
LIN {X 0,Y 545.209,Z 138.06,A -85,B 0,C 180,E1 -3600.739,E2 -3600.739} C_VEL
LIN {X 0,Y 545.17,Z 138.071,A -85,B 0,C 180,E1 -3602.956,E2 -3602.956} C_VEL
LIN {X 0,Y 545.168,Z 138.073,A -85,B 0,C 180,E1 -3605.92,E2 -3605.92} C_VEL
LIN {X 0,Y 545.114,Z 138.076,A -85,B 0,C 180,E1 -3608.901,E2 -3608.901} C_VEL
LIN {X 0,Y 545.132,Z 138.075,A -85,B 0,C 180,E1 -3611.905,E2 -3611.905} C_VEL
LIN {X 0,Y 545.083,Z 138.087,A -85,B 0,C 180,E1 -3614.944,E2 -3614.944} C_VEL
LIN {X 0,Y 545.078,Z 138.077,A -85,B 0,C 180,E1 -3618.026,E2 -3618.026} C_VEL
LIN {X 0,Y 545.092,Z 138.078,A -85,B 0,C 180,E1 -3620.373,E2 -3620.373} C_VEL
LIN {X 0,Y 545.079,Z 138.084,A -85,B 0,C 180,E1 -3623.56,E2 -3623.56} C_VEL
LIN {X 0,Y 545.078,Z 138.079,A -85,B 0,C 180,E1 -3626.001,E2 -3626.001} C_VEL
LIN {X 0,Y 545.087,Z 138.086,A -85,B 0,C 180,E1 -3628.749,E2 -3628.749} C_VEL
LIN {X 0,Y 545.058,Z 138.085,A -85,B 0,C 180,E1 -3631.68,E2 -3631.68} C_VEL
LIN {X 0,Y 545.072,Z 138.086,A -85,B 0,C 180,E1 -3634.564,E2 -3634.564} C_VEL
LIN {X 0,Y 545.034,Z 138.089,A -85,B 0,C 180,E1 -3637.305,E2 -3637.305} C_VEL
LIN {X 0,Y 545.064,Z 138.086,A -85,B 0,C 180,E1 -3640.143,E2 -3640.143} C_VEL
LIN {X 0,Y 545.078,Z 138.084,A -85,B 0,C 180,E1 -3643.107,E2 -3643.107} C_VEL
LIN {X 0,Y 545.049,Z 138.093,A -85,B 0,C 180,E1 -3646.227,E2 -3646.227} C_VEL
LIN {X 0,Y 545.081,Z 138.079,A -85,B 0,C 180,E1 -3648.886,E2 -3648.886} C_VEL
LIN {X 0,Y 545.085,Z 138.083,A -85,B 0,C 180,E1 -3650.819,E2 -3650.819} C_VEL
LIN {X 0,Y 545.043,Z 138.089,A -85,B 0,C 180,E1 -3653.62,E2 -3653.62} C_VEL
LIN {X 0,Y 545.067,Z 138.091,A -85,B 0,C 180,E1 -3656.329,E2 -3656.329} C_VEL
LIN {X 0,Y 545.069,Z 138.086,A -85,B 0,C 180,E1 -3658.953,E2 -3658.953} C_VEL
LIN {X 0,Y 545.086,Z 138.087,A -85,B 0,C 180,E1 -3661.507,E2 -3661.507} C_VEL
LIN {X 0,Y 545.15,Z 138.26,A -85,B 0,C 180,E1 -3664.528,E2 -3664.528} C_VEL
LIN {X 0,Y 545.985,Z 143.833,A -85,B 0,C 180,E1 -3665.675,E2 -3665.675} C_VEL
LIN {X 0,Y 545.679,Z 158.316,A -85,B 0,C 180,E1 -3668.466,E2 -3668.466} C_VEL
LIN {X 0,Y 545.447,Z 172.909,A -85,B 0,C 180,E1 -3671.209,E2 -3671.209} C_VEL
LIN {X 0,Y 545.244,Z 187.529,A -85,B 0,C 180,E1 -3673.911,E2 -3673.911} C_VEL
LIN {X 0,Y 545.153,Z 195.991,A -85,B 0,C 180,E1 -3675.433,E2 -3675.433} C_VEL
LIN {X 0,Y 546.512,Z 204.928,A -85,B 0,C 180,E1 -3675.613,E2 -3675.613} C_VEL
LIN {X 0,Y 546.241,Z 300.767,A -85,B 0,C 180,E1 -3676.893,E2 -3676.893} C_VEL
LIN {X 0,Y 546.131,Z 310.664,A -85,B 0,C 180,E1 -3677.104,E2 -3677.104} C_VEL
LIN {X 0,Y 546.007,Z 320.642,A -85,B 0,C 180,E1 -3677.408,E2 -3677.408} C_VEL
LIN {X 0,Y 545.829,Z 330,A -85,B 0,C 180,E1 -3677.781,E2 -3677.781} C_VEL
LIN {X 0,Y 545.661,Z 340.246,A -85,B 0,C 180,E1 -3678.302,E2 -3678.302} C_VEL
LIN {X 0,Y 545.518,Z 349.146,A -85,B 0,C 180,E1 -3678.858,E2 -3678.858} C_VEL
LIN {X 0,Y 545.367,Z 357.878,A -85,B 0,C 180,E1 -3679.512,E2 -3679.512} C_VEL
LIN {X 0,Y 545.212,Z 365.275,A -85,B 0,C 180,E1 -3680.166,E2 -3680.166} C_VEL
LIN {X 0,Y 545.046,Z 372.495,A -85,B 0,C 180,E1 -3680.912,E2 -3680.912} C_VEL
LIN {X 0,Y 544.942,Z 378.698,A -85,B 0,C 180,E1 -3681.658,E2 -3681.658} C_VEL
LIN {X 0,Y 544.836,Z 385.235,A -85,B 0,C 180,E1 -3682.589,E2 -3682.589} C_VEL
LIN {X 0,Y 544.742,Z 390.21,A -85,B 0,C 180,E1 -3683.425,E2 -3683.425} C_VEL
LIN {X 0,Y 544.739,Z 395.223,A -85,B 0,C 180,E1 -3684.447,E2 -3684.447} C_VEL
LIN {X 0,Y 544.662,Z 399.541,A -85,B 0,C 180,E1 -3685.56,E2 -3685.56} C_VEL
LIN {X 0,Y 544.669,Z 401.904,A -85,B 0,C 180,E1 -3686.301,E2 -3686.301} C_VEL
LIN {X 0,Y 544.65,Z 403.699,A -85,B 0,C 180,E1 -3687.041,E2 -3687.041} C_VEL
LIN {X 0,Y 544.546,Z 406.135,A -85,B 0,C 180,E1 -3688.521,E2 -3688.521} C_VEL
LIN {X 0,Y 544.542,Z 406.721,A -85,B 0,C 180,E1 -3689.261,E2 -3689.261} C_VEL
LIN {X 0,Y 544.542,Z 406.721,A -85,B 0,C 180,E1 -3690.739,E2 -3690.739} C_VEL
LIN {X 0,Y 544.546,Z 406.135,A -85,B 0,C 180,E1 -3691.479,E2 -3691.479} C_VEL
LIN {X 0,Y 544.65,Z 403.699,A -85,B 0,C 180,E1 -3692.959,E2 -3692.959} C_VEL
LIN {X 0,Y 544.684,Z 400.757,A -85,B 0,C 180,E1 -3694.069,E2 -3694.069} C_VEL
LIN {X 0,Y 544.653,Z 396.773,A -85,B 0,C 180,E1 -3695.182,E2 -3695.182} C_VEL
LIN {X 0,Y 544.759,Z 392.511,A -85,B 0,C 180,E1 -3696.128,E2 -3696.128} C_VEL
LIN {X 0,Y 544.79,Z 387.545,A -85,B 0,C 180,E1 -3697.039,E2 -3697.039} C_VEL
LIN {X 0,Y 544.892,Z 381.45,A -85,B 0,C 180,E1 -3697.97,E2 -3697.97} C_VEL
LIN {X 0,Y 544.991,Z 375.75,A -85,B 0,C 180,E1 -3698.715,E2 -3698.715} C_VEL
LIN {X 0,Y 545.152,Z 367.194,A -85,B 0,C 180,E1 -3699.648,E2 -3699.648} C_VEL
LIN {X 0,Y 545.344,Z 359.013,A -85,B 0,C 180,E1 -3700.394,E2 -3700.394} C_VEL
LIN {X 0,Y 545.486,Z 350.498,A -85,B 0,C 180,E1 -3701.049,E2 -3701.049} C_VEL
LIN {X 0,Y 545.665,Z 341.287,A -85,B 0,C 180,E1 -3701.638,E2 -3701.638} C_VEL
LIN {X 0,Y 545.84,Z 332.016,A -85,B 0,C 180,E1 -3702.124,E2 -3702.124} C_VEL
LIN {X 0,Y 545.944,Z 323.218,A -85,B 0,C 180,E1 -3702.499,E2 -3702.499} C_VEL
LIN {X 0,Y 546.114,Z 313.287,A -85,B 0,C 180,E1 -3702.826,E2 -3702.826} C_VEL
LIN {X 0,Y 546.179,Z 303.43,A -85,B 0,C 180,E1 -3703.061,E2 -3703.061} C_VEL
LIN {X 0,Y 546.35,Z 278.822,A -85,B 0,C 180,E1 -3703.412,E2 -3703.412} C_VEL
LIN {X 0,Y 546.373,Z 203.354,A -85,B 0,C 180,E1 -3704.411,E2 -3704.411} C_VEL
LIN {X 0,Y 545.156,Z 195.989,A -85,B 0,C 180,E1 -3704.567,E2 -3704.567} C_VEL
LIN {X 0,Y 545.324,Z 181.266,A -85,B 0,C 180,E1 -3707.242,E2 -3707.242} C_VEL
LIN {X 0,Y 545.589,Z 166.089,A -85,B 0,C 180,E1 -3710.062,E2 -3710.062} C_VEL
LIN {X 0,Y 545.915,Z 149.017,A -85,B 0,C 180,E1 -3713.32,E2 -3713.32} C_VEL
LIN {X 0,Y 545.926,Z 142.809,A -85,B 0,C 180,E1 -3714.53,E2 -3714.53} C_VEL
LIN {X 0,Y 545.129,Z 138.109,A -85,B 0,C 180,E1 -3715.527,E2 -3715.527} C_VEL
LIN {X 0,Y 545.086,Z 138.087,A -85,B 0,C 180,E1 -3718.493,E2 -3718.493} C_VEL
LIN {X 0,Y 545.069,Z 138.086,A -85,B 0,C 180,E1 -3721.047,E2 -3721.047} C_VEL
LIN {X 0,Y 545.067,Z 138.091,A -85,B 0,C 180,E1 -3723.671,E2 -3723.671} C_VEL
LIN {X 0,Y 545.071,Z 138.084,A -85,B 0,C 180,E1 -3726.926,E2 -3726.926} C_VEL
LIN {X 0,Y 545.069,Z 138.082,A -85,B 0,C 180,E1 -3730.142,E2 -3730.142} C_VEL
LIN {X 0,Y 545.078,Z 138.085,A -85,B 0,C 180,E1 -3733.106,E2 -3733.106} C_VEL
LIN {X 0,Y 545.049,Z 138.087,A -85,B 0,C 180,E1 -3736.226,E2 -3736.226} C_VEL
LIN {X 0,Y 545.08,Z 138.084,A -85,B 0,C 180,E1 -3738.885,E2 -3738.885} C_VEL
LIN {X 0,Y 545.079,Z 138.082,A -85,B 0,C 180,E1 -3740.818,E2 -3740.818} C_VEL
LIN {X 0,Y 545.041,Z 138.091,A -85,B 0,C 180,E1 -3743.619,E2 -3743.619} C_VEL
LIN {X 0,Y 545.069,Z 138.08,A -85,B 0,C 180,E1 -3746.328,E2 -3746.328} C_VEL
LIN {X 0,Y 545.066,Z 138.089,A -85,B 0,C 180,E1 -3748.952,E2 -3748.952} C_VEL
LIN {X 0,Y 545.099,Z 138.08,A -85,B 0,C 180,E1 -3751.507,E2 -3751.507} C_VEL
LIN {X 0,Y 545.093,Z 138.079,A -85,B 0,C 180,E1 -3754.491,E2 -3754.491} C_VEL
LIN {X 0,Y 545.036,Z 138.093,A -85,B 0,C 180,E1 -3757.242,E2 -3757.242} C_VEL
LIN {X 0,Y 545.118,Z 138.076,A -85,B 0,C 180,E1 -3760.414,E2 -3760.414} C_VEL
LIN {X 0,Y 545.07,Z 138.083,A -85,B 0,C 180,E1 -3763.521,E2 -3763.521} C_VEL
LIN {X 0,Y 545.093,Z 138.08,A -85,B 0,C 180,E1 -3765.82,E2 -3765.82} C_VEL
LIN {X 0,Y 545.114,Z 138.078,A -85,B 0,C 180,E1 -3768.849,E2 -3768.849} C_VEL
LIN {X 0,Y 545.125,Z 138.073,A -85,B 0,C 180,E1 -3771.847,E2 -3771.847} C_VEL
LIN {X 0,Y 545.201,Z 138.072,A -85,B 0,C 180,E1 -3774.823,E2 -3774.823} C_VEL
LIN {X 0,Y 545.191,Z 138.068,A -85,B 0,C 180,E1 -3777.783,E2 -3777.783} C_VEL
LIN {X 0,Y 545.21,Z 138.065,A -85,B 0,C 180,E1 -3780.738,E2 -3780.738} C_VEL
LIN {X 0,Y 545.169,Z 138.071,A -85,B 0,C 180,E1 -3782.955,E2 -3782.955} C_VEL
LIN {X 0,Y 545.167,Z 138.076,A -85,B 0,C 180,E1 -3785.919,E2 -3785.919} C_VEL
LIN {X 0,Y 545.114,Z 138.073,A -85,B 0,C 180,E1 -3788.9,E2 -3788.9} C_VEL
LIN {X 0,Y 545.131,Z 138.078,A -85,B 0,C 180,E1 -3791.904,E2 -3791.904} C_VEL
LIN {X 0,Y 545.081,Z 138.082,A -85,B 0,C 180,E1 -3794.943,E2 -3794.943} C_VEL
LIN {X 0,Y 545.078,Z 138.083,A -85,B 0,C 180,E1 -3798.025,E2 -3798.025} C_VEL
LIN {X 0,Y 545.09,Z 138.081,A -85,B 0,C 180,E1 -3800.372,E2 -3800.372} C_VEL
LIN {X 0,Y 545.087,Z 138.088,A -85,B 0,C 180,E1 -3803.559,E2 -3803.559} C_VEL
LIN {X 0,Y 545.084,Z 138.082,A -85,B 0,C 180,E1 -3806,E2 -3806} C_VEL
LIN {X 0,Y 545.085,Z 138.08,A -85,B 0,C 180,E1 -3808.748,E2 -3808.748} C_VEL
LIN {X 0,Y 545.073,Z 138.09,A -85,B 0,C 180,E1 -3811.682,E2 -3811.682} C_VEL
LIN {X 0,Y 545.08,Z 138.078,A -85,B 0,C 180,E1 -3814.563,E2 -3814.563} C_VEL
LIN {X 0,Y 545.061,Z 138.088,A -85,B 0,C 180,E1 -3817,E2 -3817} C_VEL
LIN {X 0,Y 544.353,Z 138.182,A -85,B 0,C 180,E1 -3817.617,E2 -3817.617} C_VEL
LIN {X 0,Y 541.489,Z 138.536,A -85,B 0,C 180,E1 -3818.618,E2 -3818.618} C_VEL
LIN {X 0,Y 539.103,Z 138.832,A -85,B 0,C 180,E1 -3819.423,E2 -3819.423} C_VEL
LIN {X 0,Y 538.093,Z 138.951,A -85,B 0,C 180,E1 -3820.045,E2 -3820.045} C_VEL
LIN {X 0,Y 538.016,Z 138.959,A -85,B 0,C 180,E1 -3820.256,E2 -3820.256} C_VEL
LIN {X 0,Y 538.029,Z 138.966,A -85,B 0,C 180,E1 -3822.988,E2 -3822.988} C_VEL
LIN {X 0,Y 538.024,Z 138.957,A -85,B 0,C 180,E1 -3825.925,E2 -3825.925} C_VEL
LIN {X 0,Y 538.047,Z 138.96,A -85,B 0,C 180,E1 -3829.252,E2 -3829.252} C_VEL
LIN {X 0,Y 537.99,Z 138.967,A -85,B 0,C 180,E1 -3832.123,E2 -3832.123} C_VEL
LIN {X 0,Y 538.015,Z 138.963,A -85,B 0,C 180,E1 -3834.917,E2 -3834.917} C_VEL
LIN {X 0,Y 538.027,Z 138.962,A -85,B 0,C 180,E1 -3837.618,E2 -3837.618} C_VEL
LIN {X 0,Y 538.039,Z 138.96,A -85,B 0,C 180,E1 -3840.241,E2 -3840.241} C_VEL
LIN {X 0,Y 538.061,Z 138.966,A -85,B 0,C 180,E1 -3842.796,E2 -3842.796} C_VEL
LIN {X 0,Y 538.045,Z 138.961,A -85,B 0,C 180,E1 -3845.293,E2 -3845.293} C_VEL
LIN {X 0,Y 538.012,Z 138.966,A -85,B 0,C 180,E1 -3848.042,E2 -3848.042} C_VEL
LIN {X 0,Y 538.034,Z 138.965,A -85,B 0,C 180,E1 -3850.94,E2 -3850.94} C_VEL
LIN {X 0,Y 538.021,Z 138.963,A -85,B 0,C 180,E1 -3853.299,E2 -3853.299} C_VEL
LIN {X 0,Y 538.061,Z 138.959,A -85,B 0,C 180,E1 -3855.631,E2 -3855.631} C_VEL
LIN {X 0,Y 538.075,Z 138.96,A -85,B 0,C 180,E1 -3858.702,E2 -3858.702} C_VEL
LIN {X 0,Y 538.084,Z 138.959,A -85,B 0,C 180,E1 -3861.74,E2 -3861.74} C_VEL
LIN {X 0,Y 538.16,Z 138.948,A -85,B 0,C 180,E1 -3864.755,E2 -3864.755} C_VEL
LIN {X 0,Y 538.167,Z 138.95,A -85,B 0,C 180,E1 -3867.755,E2 -3867.755} C_VEL
LIN {X 0,Y 538.18,Z 138.944,A -85,B 0,C 180,E1 -3870.748,E2 -3870.748} C_VEL
LIN {X 0,Y 538.136,Z 138.949,A -85,B 0,C 180,E1 -3872.994,E2 -3872.994} C_VEL
LIN {X 0,Y 538.123,Z 138.957,A -85,B 0,C 180,E1 -3875.997,E2 -3875.997} C_VEL
LIN {X 0,Y 538.069,Z 138.958,A -85,B 0,C 180,E1 -3879.018,E2 -3879.018} C_VEL
LIN {X 0,Y 538.08,Z 138.96,A -85,B 0,C 180,E1 -3882.062,E2 -3882.062} C_VEL
LIN {X 0,Y 538.042,Z 138.964,A -85,B 0,C 180,E1 -3885.144,E2 -3885.144} C_VEL
LIN {X 0,Y 538.028,Z 138.963,A -85,B 0,C 180,E1 -3888.27,E2 -3888.27} C_VEL
LIN {X 0,Y 538.036,Z 138.962,A -85,B 0,C 180,E1 -3890.651,E2 -3890.651} C_VEL
LIN {X 0,Y 538.021,Z 138.965,A -85,B 0,C 180,E1 -3893.887,E2 -3893.887} C_VEL
LIN {X 0,Y 538.038,Z 138.961,A -85,B 0,C 180,E1 -3896.367,E2 -3896.367} C_VEL
LIN {X 0,Y 538.053,Z 138.962,A -85,B 0,C 180,E1 -3898.939,E2 -3898.939} C_VEL
LIN {X 0,Y 538.023,Z 138.963,A -85,B 0,C 180,E1 -3901.89,E2 -3901.89} C_VEL
LIN {X 0,Y 538.022,Z 138.96,A -85,B 0,C 180,E1 -3904.62,E2 -3904.62} C_VEL
LIN {X 0,Y 538.003,Z 138.972,A -85,B 0,C 180,E1 -3907.17,E2 -3907.17} C_VEL
LIN {X 0,Y 538.025,Z 138.959,A -85,B 0,C 180,E1 -3909.796,E2 -3909.796} C_VEL
LIN {X 0,Y 538.014,Z 138.958,A -85,B 0,C 180,E1 -3912.786,E2 -3912.786} C_VEL
LIN {X 0,Y 538.027,Z 138.965,A -85,B 0,C 180,E1 -3915.141,E2 -3915.141} C_VEL
LIN {X 0,Y 538.036,Z 138.962,A -85,B 0,C 180,E1 -3918.228,E2 -3918.228} C_VEL
LIN {X 0,Y 538.01,Z 138.966,A -85,B 0,C 180,E1 -3921.17,E2 -3921.17} C_VEL
LIN {X 0,Y 538.025,Z 138.964,A -85,B 0,C 180,E1 -3924.083,E2 -3924.083} C_VEL
LIN {X 0,Y 538.031,Z 138.966,A -85,B 0,C 180,E1 -3926.728,E2 -3926.728} C_VEL
LIN {X 0,Y 538.021,Z 138.962,A -85,B 0,C 180,E1 -3929.556,E2 -3929.556} C_VEL
LIN {X 0,Y 538.043,Z 138.96,A -85,B 0,C 180,E1 -3931.951,E2 -3931.951} C_VEL
LIN {X 0,Y 538.071,Z 138.961,A -85,B 0,C 180,E1 -3934.468,E2 -3934.468} C_VEL
LIN {X 0,Y 538.018,Z 138.963,A -85,B 0,C 180,E1 -3936.929,E2 -3936.929} C_VEL
LIN {X 0,Y 538.074,Z 138.956,A -85,B 0,C 180,E1 -3940.148,E2 -3940.148} C_VEL
LIN {X 0,Y 538.02,Z 138.96,A -85,B 0,C 180,E1 -3943.299,E2 -3943.299} C_VEL
LIN {X 0,Y 538.06,Z 138.961,A -85,B 0,C 180,E1 -3945.631,E2 -3945.631} C_VEL
LIN {X 0,Y 538.072,Z 138.951,A -85,B 0,C 180,E1 -3948.702,E2 -3948.702} C_VEL
LIN {X 0,Y 538.082,Z 138.955,A -85,B 0,C 180,E1 -3951.74,E2 -3951.74} C_VEL
LIN {X 0,Y 538.158,Z 138.945,A -85,B 0,C 180,E1 -3954.755,E2 -3954.755} C_VEL
LIN {X 0,Y 538.163,Z 138.947,A -85,B 0,C 180,E1 -3957.755,E2 -3957.755} C_VEL
LIN {X 0,Y 538.179,Z 138.935,A -85,B 0,C 180,E1 -3960.749,E2 -3960.749} C_VEL
LIN {X 0,Y 538.136,Z 138.948,A -85,B 0,C 180,E1 -3962.995,E2 -3962.995} C_VEL
LIN {X 0,Y 538.121,Z 138.95,A -85,B 0,C 180,E1 -3965.998,E2 -3965.998} C_VEL
LIN {X 0,Y 538.065,Z 138.955,A -85,B 0,C 180,E1 -3969.018,E2 -3969.018} C_VEL
LIN {X 0,Y 538.081,Z 138.953,A -85,B 0,C 180,E1 -3972.063,E2 -3972.063} C_VEL
LIN {X 0,Y 538.043,Z 138.967,A -85,B 0,C 180,E1 -3975.144,E2 -3975.144} C_VEL
LIN {X 0,Y 538.031,Z 138.954,A -85,B 0,C 180,E1 -3978.271,E2 -3978.271} C_VEL
LIN {X 0,Y 538.037,Z 138.959,A -85,B 0,C 180,E1 -3980.652,E2 -3980.652} C_VEL
LIN {X 0,Y 538.002,Z 138.964,A -85,B 0,C 180,E1 -3983.889,E2 -3983.889} C_VEL
LIN {X 0,Y 538.04,Z 138.957,A -85,B 0,C 180,E1 -3986.367,E2 -3986.367} C_VEL
LIN {X 0,Y 538.029,Z 138.968,A -85,B 0,C 180,E1 -3988.934,E2 -3988.934} C_VEL
LIN {X 0,Y 538.013,Z 138.963,A -85,B 0,C 180,E1 -3991.889,E2 -3991.889} C_VEL
LIN {X 0,Y 538.021,Z 138.965,A -85,B 0,C 180,E1 -3994.62,E2 -3994.62} C_VEL
LIN {X 0,Y 538.003,Z 138.966,A -85,B 0,C 180,E1 -3997.17,E2 -3997.17} C_VEL
LIN {X 0,Y 538.021,Z 138.96,A -85,B 0,C 180,E1 -3999.798,E2 -3999.798} C_VEL
LIN {X 0,Y 538.018,Z 138.967,A -85,B 0,C 180,E1 -4002.787,E2 -4002.787} C_VEL
LIN {X 0,Y 538.019,Z 138.964,A -85,B 0,C 180,E1 -4005.927,E2 -4005.927} C_VEL
LIN {X 0,Y 538.03,Z 138.968,A -85,B 0,C 180,E1 -4008.227,E2 -4008.227} C_VEL
LIN {X 0,Y 538.016,Z 138.962,A -85,B 0,C 180,E1 -4011.17,E2 -4011.17} C_VEL
LIN {X 0,Y 537.995,Z 138.97,A -85,B 0,C 180,E1 -4014.089,E2 -4014.089} C_VEL
LIN {X 0,Y 538.032,Z 138.962,A -85,B 0,C 180,E1 -4016.728,E2 -4016.728} C_VEL
LIN {X 0,Y 538.028,Z 138.966,A -85,B 0,C 180,E1 -4019.557,E2 -4019.557} C_VEL
LIN {X 0,Y 538.058,Z 138.963,A -85,B 0,C 180,E1 -4022.649,E2 -4022.649} C_VEL
LIN {X 0,Y 538.099,Z 139.11,A -85,B 0,C 180,E1 -4024.359,E2 -4024.359} C_VEL
LIN {X 0,Y 539.036,Z 145.333,A -85,B 0,C 180,E1 -4025.663,E2 -4025.663} C_VEL
LIN {X 0,Y 538.683,Z 160.249,A -85,B 0,C 180,E1 -4028.574,E2 -4028.574} C_VEL
LIN {X 0,Y 538.45,Z 173.823,A -85,B 0,C 180,E1 -4031.153,E2 -4031.153} C_VEL
LIN {X 0,Y 538.197,Z 189.441,A -85,B 0,C 180,E1 -4034.084,E2 -4034.084} C_VEL
LIN {X 0,Y 538.121,Z 195.572,A -85,B 0,C 180,E1 -4035.221,E2 -4035.221} C_VEL
LIN {X 0,Y 538.545,Z 198.62,A -85,B 0,C 180,E1 -4035.314,E2 -4035.314} C_VEL
LIN {X 0,Y 539.659,Z 205.936,A -85,B 0,C 180,E1 -4035.443,E2 -4035.443} C_VEL
LIN {X 0,Y 539.34,Z 300.576,A -85,B 0,C 180,E1 -4036.723,E2 -4036.723} C_VEL
LIN {X 0,Y 539.228,Z 310.472,A -85,B 0,C 180,E1 -4036.936,E2 -4036.936} C_VEL
LIN {X 0,Y 539.069,Z 320.45,A -85,B 0,C 180,E1 -4037.243,E2 -4037.243} C_VEL
LIN {X 0,Y 538.897,Z 329.808,A -85,B 0,C 180,E1 -4037.622,E2 -4037.622} C_VEL
LIN {X 0,Y 538.725,Z 339.491,A -85,B 0,C 180,E1 -4038.116,E2 -4038.116} C_VEL
LIN {X 0,Y 538.525,Z 348.954,A -85,B 0,C 180,E1 -4038.711,E2 -4038.711} C_VEL
LIN {X 0,Y 538.342,Z 357.685,A -85,B 0,C 180,E1 -4039.374,E2 -4039.374} C_VEL
LIN {X 0,Y 538.166,Z 365.082,A -85,B 0,C 180,E1 -4040.036,E2 -4040.036} C_VEL
LIN {X 0,Y 538.003,Z 372.303,A -85,B 0,C 180,E1 -4040.792,E2 -4040.792} C_VEL
LIN {X 0,Y 537.9,Z 378.506,A -85,B 0,C 180,E1 -4041.548,E2 -4041.548} C_VEL
LIN {X 0,Y 537.754,Z 385.042,A -85,B 0,C 180,E1 -4042.491,E2 -4042.491} C_VEL
LIN {X 0,Y 537.641,Z 390.583,A -85,B 0,C 180,E1 -4043.449,E2 -4043.449} C_VEL
LIN {X 0,Y 537.653,Z 395.031,A -85,B 0,C 180,E1 -4044.374,E2 -4044.374} C_VEL
LIN {X 0,Y 537.558,Z 399.349,A -85,B 0,C 180,E1 -4045.501,E2 -4045.501} C_VEL
LIN {X 0,Y 537.591,Z 401.713,A -85,B 0,C 180,E1 -4046.252,E2 -4046.252} C_VEL
LIN {X 0,Y 537.551,Z 403.507,A -85,B 0,C 180,E1 -4047.002,E2 -4047.002} C_VEL
LIN {X 0,Y 537.451,Z 405.943,A -85,B 0,C 180,E1 -4048.501,E2 -4048.501} C_VEL
LIN {X 0,Y 537.444,Z 406.53,A -85,B 0,C 180,E1 -4049.251,E2 -4049.251} C_VEL
LIN {X 0,Y 537.444,Z 406.53,A -85,B 0,C 180,E1 -4050.749,E2 -4050.749} C_VEL
LIN {X 0,Y 537.451,Z 405.943,A -85,B 0,C 180,E1 -4051.499,E2 -4051.499} C_VEL
LIN {X 0,Y 537.551,Z 403.507,A -85,B 0,C 180,E1 -4052.998,E2 -4052.998} C_VEL
LIN {X 0,Y 537.604,Z 400.565,A -85,B 0,C 180,E1 -4054.123,E2 -4054.123} C_VEL
LIN {X 0,Y 537.586,Z 396.582,A -85,B 0,C 180,E1 -4055.251,E2 -4055.251} C_VEL
LIN {X 0,Y 537.625,Z 391.788,A -85,B 0,C 180,E1 -4056.314,E2 -4056.314} C_VEL
LIN {X 0,Y 537.754,Z 386.198,A -85,B 0,C 180,E1 -4057.321,E2 -4057.321} C_VEL
LIN {X 0,Y 537.867,Z 379.882,A -85,B 0,C 180,E1 -4058.264,E2 -4058.264} C_VEL
LIN {X 0,Y 537.952,Z 373.93,A -85,B 0,C 180,E1 -4059.019,E2 -4059.019} C_VEL
LIN {X 0,Y 538.112,Z 367.002,A -85,B 0,C 180,E1 -4059.775,E2 -4059.775} C_VEL
LIN {X 0,Y 538.332,Z 358.821,A -85,B 0,C 180,E1 -4060.531,E2 -4060.531} C_VEL
LIN {X 0,Y 538.499,Z 350.306,A -85,B 0,C 180,E1 -4061.194,E2 -4061.194} C_VEL
LIN {X 0,Y 538.647,Z 342.109,A -85,B 0,C 180,E1 -4061.732,E2 -4061.732} C_VEL
LIN {X 0,Y 538.872,Z 332.832,A -85,B 0,C 180,E1 -4062.236,E2 -4062.236} C_VEL
LIN {X 0,Y 539.016,Z 323.026,A -85,B 0,C 180,E1 -4062.663,E2 -4062.663} C_VEL
LIN {X 0,Y 539.202,Z 313.096,A -85,B 0,C 180,E1 -4062.993,E2 -4062.993} C_VEL
LIN {X 0,Y 539.266,Z 303.238,A -85,B 0,C 180,E1 -4063.231,E2 -4063.231} C_VEL
LIN {X 0,Y 539.452,Z 278.63,A -85,B 0,C 180,E1 -4063.586,E2 -4063.586} C_VEL
LIN {X 0,Y 539.569,Z 204.567,A -85,B 0,C 180,E1 -4064.578,E2 -4064.578} C_VEL
LIN {X 0,Y 538.124,Z 195.799,A -85,B 0,C 180,E1 -4064.761,E2 -4064.761} C_VEL
LIN {X 0,Y 538.159,Z 191.559,A -85,B 0,C 180,E1 -4065.528,E2 -4065.528} C_VEL
LIN {X 0,Y 538.4,Z 175.913,A -85,B 0,C 180,E1 -4068.454,E2 -4068.454} C_VEL
LIN {X 0,Y 538.631,Z 162.319,A -85,B 0,C 180,E1 -4071.027,E2 -4071.027} C_VEL
LIN {X 0,Y 538.981,Z 147.849,A -85,B 0,C 180,E1 -4073.842,E2 -4073.842} C_VEL
LIN {X 0,Y 538.766,Z 142.67,A -85,B 0,C 180,E1 -4074.878,E2 -4074.878} C_VEL
LIN {X 0,Y 538.077,Z 138.987,A -85,B 0,C 180,E1 -4075.698,E2 -4075.698} C_VEL
LIN {X 0,Y 538.036,Z 138.967,A -85,B 0,C 180,E1 -4078.05,E2 -4078.05} C_VEL
LIN {X 0,Y 538.023,Z 138.965,A -85,B 0,C 180,E1 -4080.626,E2 -4080.626} C_VEL
LIN {X 0,Y 538.047,Z 138.961,A -85,B 0,C 180,E1 -4083.282,E2 -4083.282} C_VEL
LIN {X 0,Y 537.995,Z 138.971,A -85,B 0,C 180,E1 -4086.004,E2 -4086.004} C_VEL
LIN {X 0,Y 538.016,Z 138.962,A -85,B 0,C 180,E1 -4088.83,E2 -4088.83} C_VEL
LIN {X 0,Y 538.03,Z 138.967,A -85,B 0,C 180,E1 -4091.773,E2 -4091.773} C_VEL
LIN {X 0,Y 538.006,Z 138.964,A -85,B 0,C 180,E1 -4094.862,E2 -4094.862} C_VEL
LIN {X 0,Y 538.018,Z 138.967,A -85,B 0,C 180,E1 -4097.213,E2 -4097.213} C_VEL
LIN {X 0,Y 538.021,Z 138.96,A -85,B 0,C 180,E1 -4100.202,E2 -4100.202} C_VEL
LIN {X 0,Y 538.023,Z 138.967,A -85,B 0,C 180,E1 -4103.067,E2 -4103.067} C_VEL
LIN {X 0,Y 538.022,Z 138.959,A -85,B 0,C 180,E1 -4105.827,E2 -4105.827} C_VEL
LIN {X 0,Y 538.009,Z 138.964,A -85,B 0,C 180,E1 -4108.498,E2 -4108.498} C_VEL
LIN {X 0,Y 538.058,Z 138.964,A -85,B 0,C 180,E1 -4111.099,E2 -4111.099} C_VEL
LIN {X 0,Y 538.04,Z 138.957,A -85,B 0,C 180,E1 -4113.633,E2 -4113.633} C_VEL
LIN {X 0,Y 538.004,Z 138.963,A -85,B 0,C 180,E1 -4116.121,E2 -4116.121} C_VEL
LIN {X 0,Y 538.037,Z 138.959,A -85,B 0,C 180,E1 -4119.348,E2 -4119.348} C_VEL
LIN {X 0,Y 538.052,Z 138.956,A -85,B 0,C 180,E1 -4122.517,E2 -4122.517} C_VEL
LIN {X 0,Y 538.062,Z 138.956,A -85,B 0,C 180,E1 -4125.63,E2 -4125.63} C_VEL
LIN {X 0,Y 538.074,Z 138.957,A -85,B 0,C 180,E1 -4128.701,E2 -4128.701} C_VEL
LIN {X 0,Y 538.082,Z 138.949,A -85,B 0,C 180,E1 -4131.739,E2 -4131.739} C_VEL
LIN {X 0,Y 538.158,Z 138.95,A -85,B 0,C 180,E1 -4134.755,E2 -4134.755} C_VEL
LIN {X 0,Y 538.163,Z 138.943,A -85,B 0,C 180,E1 -4137.754,E2 -4137.754} C_VEL
LIN {X 0,Y 538.18,Z 138.94,A -85,B 0,C 180,E1 -4140.748,E2 -4140.748} C_VEL
LIN {X 0,Y 538.135,Z 138.947,A -85,B 0,C 180,E1 -4142.994,E2 -4142.994} C_VEL
LIN {X 0,Y 538.12,Z 138.955,A -85,B 0,C 180,E1 -4145.997,E2 -4145.997} C_VEL
LIN {X 0,Y 538.065,Z 138.95,A -85,B 0,C 180,E1 -4149.017,E2 -4149.017} C_VEL
LIN {X 0,Y 538.079,Z 138.959,A -85,B 0,C 180,E1 -4152.062,E2 -4152.062} C_VEL
LIN {X 0,Y 538.041,Z 138.96,A -85,B 0,C 180,E1 -4155.143,E2 -4155.143} C_VEL
LIN {X 0,Y 538.03,Z 138.957,A -85,B 0,C 180,E1 -4158.27,E2 -4158.27} C_VEL
LIN {X 0,Y 538.034,Z 138.958,A -85,B 0,C 180,E1 -4160.651,E2 -4160.651} C_VEL
LIN {X 0,Y 538.019,Z 138.968,A -85,B 0,C 180,E1 -4163.887,E2 -4163.887} C_VEL
LIN {X 0,Y 538.045,Z 138.955,A -85,B 0,C 180,E1 -4166.366,E2 -4166.366} C_VEL
LIN {X 0,Y 538.026,Z 138.96,A -85,B 0,C 180,E1 -4168.934,E2 -4168.934} C_VEL
LIN {X 0,Y 538.023,Z 138.965,A -85,B 0,C 180,E1 -4171.89,E2 -4171.89} C_VEL
LIN {X 0,Y 538.029,Z 138.956,A -85,B 0,C 180,E1 -4174.621,E2 -4174.621} C_VEL
LIN {X 0,Y 538.003,Z 138.969,A -85,B 0,C 180,E1 -4177.17,E2 -4177.17} C_VEL
LIN {X 0,Y 538.016,Z 138.959,A -85,B 0,C 180,E1 -4180.256,E2 -4180.256} C_VEL
LIN {X 0,Y 537.367,Z 139.044,A -85,B 0,C 180,E1 -4180.881,E2 -4180.881} C_VEL
LIN {X 0,Y 534.519,Z 139.404,A -85,B 0,C 180,E1 -4181.896,E2 -4181.896} C_VEL
LIN {X 0,Y 532.097,Z 139.709,A -85,B 0,C 180,E1 -4182.713,E2 -4182.713} C_VEL
LIN {X 0,Y 531.049,Z 139.838,A -85,B 0,C 180,E1 -4183.344,E2 -4183.344} C_VEL
LIN {X 0,Y 530.96,Z 139.846,A -85,B 0,C 180,E1 -4183.558,E2 -4183.558} C_VEL
LIN {X 0,Y 530.959,Z 139.838,A -85,B 0,C 180,E1 -4186.505,E2 -4186.505} C_VEL
LIN {X 0,Y 530.98,Z 139.839,A -85,B 0,C 180,E1 -4189.567,E2 -4189.567} C_VEL
LIN {X 0,Y 530.965,Z 139.845,A -85,B 0,C 180,E1 -4192.577,E2 -4192.577} C_VEL
LIN {X 0,Y 530.997,Z 139.835,A -85,B 0,C 180,E1 -4195.311,E2 -4195.311} C_VEL
LIN {X 0,Y 530.978,Z 139.84,A -85,B 0,C 180,E1 -4198.033,E2 -4198.033} C_VEL
LIN {X 0,Y 530.992,Z 139.84,A -85,B 0,C 180,E1 -4200.873,E2 -4200.873} C_VEL
LIN {X 0,Y 531.001,Z 139.839,A -85,B 0,C 180,E1 -4203.256,E2 -4203.256} C_VEL
LIN {X 0,Y 530.993,Z 139.839,A -85,B 0,C 180,E1 -4205.958,E2 -4205.958} C_VEL
LIN {X 0,Y 530.997,Z 139.841,A -85,B 0,C 180,E1 -4209.062,E2 -4209.062} C_VEL
LIN {X 0,Y 531.013,Z 139.843,A -85,B 0,C 180,E1 -4212.278,E2 -4212.278} C_VEL
LIN {X 0,Y 531.016,Z 139.836,A -85,B 0,C 180,E1 -4215.436,E2 -4215.436} C_VEL
LIN {X 0,Y 531.034,Z 139.84,A -85,B 0,C 180,E1 -4218.55,E2 -4218.55} C_VEL
LIN {X 0,Y 531.054,Z 139.834,A -85,B 0,C 180,E1 -4221.63,E2 -4221.63} C_VEL
LIN {X 0,Y 531.119,Z 139.826,A -85,B 0,C 180,E1 -4224.685,E2 -4224.685} C_VEL
LIN {X 0,Y 531.139,Z 139.826,A -85,B 0,C 180,E1 -4227.725,E2 -4227.725} C_VEL
LIN {X 0,Y 531.15,Z 139.82,A -85,B 0,C 180,E1 -4230.758,E2 -4230.758} C_VEL
LIN {X 0,Y 531.103,Z 139.826,A -85,B 0,C 180,E1 -4233.034,E2 -4233.034} C_VEL
LIN {X 0,Y 531.083,Z 139.833,A -85,B 0,C 180,E1 -4236.077,E2 -4236.077} C_VEL
LIN {X 0,Y 531.029,Z 139.836,A -85,B 0,C 180,E1 -4239.138,E2 -4239.138} C_VEL
LIN {X 0,Y 531.038,Z 139.836,A -85,B 0,C 180,E1 -4242.225,E2 -4242.225} C_VEL
LIN {X 0,Y 530.992,Z 139.845,A -85,B 0,C 180,E1 -4245.35,E2 -4245.35} C_VEL
LIN {X 0,Y 530.987,Z 139.84,A -85,B 0,C 180,E1 -4248.521,E2 -4248.521} C_VEL
LIN {X 0,Y 530.996,Z 139.841,A -85,B 0,C 180,E1 -4250.938,E2 -4250.938} C_VEL
LIN {X 0,Y 530.976,Z 139.841,A -85,B 0,C 180,E1 -4254.224,E2 -4254.224} C_VEL
LIN {X 0,Y 531.002,Z 139.839,A -85,B 0,C 180,E1 -4256.743,E2 -4256.743} C_VEL
LIN {X 0,Y 530.997,Z 139.839,A -85,B 0,C 180,E1 -4259.321,E2 -4259.321} C_VEL
LIN {X 0,Y 530.976,Z 139.84,A -85,B 0,C 180,E1 -4262.103,E2 -4262.103} C_VEL
LIN {X 0,Y 530.979,Z 139.838,A -85,B 0,C 180,E1 -4264.853,E2 -4264.853} C_VEL
LIN {X 0,Y 530.962,Z 139.844,A -85,B 0,C 180,E1 -4267.507,E2 -4267.507} C_VEL
LIN {X 0,Y 530.98,Z 139.839,A -85,B 0,C 180,E1 -4270.433,E2 -4270.433} C_VEL
LIN {X 0,Y 530.959,Z 139.838,A -85,B 0,C 180,E1 -4273.495,E2 -4273.495} C_VEL
LIN {X 0,Y 530.963,Z 139.846,A -85,B 0,C 180,E1 -4276.506,E2 -4276.506} C_VEL
LIN {X 0,Y 530.98,Z 139.836,A -85,B 0,C 180,E1 -4279.568,E2 -4279.568} C_VEL
LIN {X 0,Y 530.964,Z 139.85,A -85,B 0,C 180,E1 -4282.577,E2 -4282.577} C_VEL
LIN {X 0,Y 530.999,Z 139.831,A -85,B 0,C 180,E1 -4285.311,E2 -4285.311} C_VEL
LIN {X 0,Y 530.978,Z 139.842,A -85,B 0,C 180,E1 -4288.033,E2 -4288.033} C_VEL
LIN {X 0,Y 530.984,Z 139.838,A -85,B 0,C 180,E1 -4290.874,E2 -4290.874} C_VEL
LIN {X 0,Y 531.007,Z 139.83,A -85,B 0,C 180,E1 -4293.257,E2 -4293.257} C_VEL
LIN {X 0,Y 530.992,Z 139.841,A -85,B 0,C 180,E1 -4295.958,E2 -4295.958} C_VEL
LIN {X 0,Y 530.995,Z 139.834,A -85,B 0,C 180,E1 -4299.062,E2 -4299.062} C_VEL
LIN {X 0,Y 531.012,Z 139.839,A -85,B 0,C 180,E1 -4302.278,E2 -4302.278} C_VEL
LIN {X 0,Y 531.015,Z 139.836,A -85,B 0,C 180,E1 -4305.436,E2 -4305.436} C_VEL
LIN {X 0,Y 531.032,Z 139.828,A -85,B 0,C 180,E1 -4308.55,E2 -4308.55} C_VEL
LIN {X 0,Y 531.051,Z 139.829,A -85,B 0,C 180,E1 -4311.63,E2 -4311.63} C_VEL
LIN {X 0,Y 531.117,Z 139.822,A -85,B 0,C 180,E1 -4314.686,E2 -4314.686} C_VEL
LIN {X 0,Y 531.135,Z 139.822,A -85,B 0,C 180,E1 -4317.725,E2 -4317.725} C_VEL
LIN {X 0,Y 531.15,Z 139.811,A -85,B 0,C 180,E1 -4320.759,E2 -4320.759} C_VEL
LIN {X 0,Y 531.103,Z 139.824,A -85,B 0,C 180,E1 -4323.035,E2 -4323.035} C_VEL
LIN {X 0,Y 531.08,Z 139.827,A -85,B 0,C 180,E1 -4326.078,E2 -4326.078} C_VEL
LIN {X 0,Y 531.025,Z 139.833,A -85,B 0,C 180,E1 -4329.139,E2 -4329.139} C_VEL
LIN {X 0,Y 531.038,Z 139.829,A -85,B 0,C 180,E1 -4332.225,E2 -4332.225} C_VEL
LIN {X 0,Y 530.993,Z 139.842,A -85,B 0,C 180,E1 -4335.35,E2 -4335.35} C_VEL
LIN {X 0,Y 530.989,Z 139.832,A -85,B 0,C 180,E1 -4338.522,E2 -4338.522} C_VEL
LIN {X 0,Y 530.997,Z 139.839,A -85,B 0,C 180,E1 -4340.938,E2 -4340.938} C_VEL
LIN {X 0,Y 530.97,Z 139.84,A -85,B 0,C 180,E1 -4344.225,E2 -4344.225} C_VEL
LIN {X 0,Y 531,Z 139.838,A -85,B 0,C 180,E1 -4346.744,E2 -4346.744} C_VEL
LIN {X 0,Y 530.981,Z 139.841,A -85,B 0,C 180,E1 -4349.323,E2 -4349.323} C_VEL
LIN {X 0,Y 530.969,Z 139.841,A -85,B 0,C 180,E1 -4352.102,E2 -4352.102} C_VEL
LIN {X 0,Y 530.976,Z 139.844,A -85,B 0,C 180,E1 -4354.853,E2 -4354.853} C_VEL
LIN {X 0,Y 530.964,Z 139.841,A -85,B 0,C 180,E1 -4357.508,E2 -4357.508} C_VEL
LIN {X 0,Y 530.98,Z 139.843,A -85,B 0,C 180,E1 -4360.434,E2 -4360.434} C_VEL
LIN {X 0,Y 530.96,Z 139.842,A -85,B 0,C 180,E1 -4363.282,E2 -4363.282} C_VEL
LIN {X 0,Y 530.976,Z 139.839,A -85,B 0,C 180,E1 -4365.623,E2 -4365.623} C_VEL
LIN {X 0,Y 530.993,Z 139.837,A -85,B 0,C 180,E1 -4368.565,E2 -4368.565} C_VEL
LIN {X 0,Y 530.96,Z 139.842,A -85,B 0,C 180,E1 -4371.53,E2 -4371.53} C_VEL
LIN {X 0,Y 530.955,Z 139.845,A -85,B 0,C 180,E1 -4374.38,E2 -4374.38} C_VEL
LIN {X 0,Y 530.968,Z 139.841,A -85,B 0,C 180,E1 -4377.134,E2 -4377.134} C_VEL
LIN {X 0,Y 530.971,Z 139.848,A -85,B 0,C 180,E1 -4379.804,E2 -4379.804} C_VEL
LIN {X 0,Y 531.016,Z 139.84,A -85,B 0,C 180,E1 -4382.468,E2 -4382.468} C_VEL
LIN {X 0,Y 531.053,Z 139.997,A -85,B 0,C 180,E1 -4384.197,E2 -4384.197} C_VEL
LIN {X 0,Y 532.026,Z 145.589,A -85,B 0,C 180,E1 -4385.4,E2 -4385.4} C_VEL
LIN {X 0,Y 531.775,Z 157.116,A -85,B 0,C 180,E1 -4387.689,E2 -4387.689} C_VEL
LIN {X 0,Y 531.539,Z 171.602,A -85,B 0,C 180,E1 -4390.497,E2 -4390.497} C_VEL
LIN {X 0,Y 531.208,Z 187.216,A -85,B 0,C 180,E1 -4393.474,E2 -4393.474} C_VEL
LIN {X 0,Y 531.097,Z 195.364,A -85,B 0,C 180,E1 -4395.019,E2 -4395.019} C_VEL
LIN {X 0,Y 531.46,Z 198.15,A -85,B 0,C 180,E1 -4395.11,E2 -4395.11} C_VEL
LIN {X 0,Y 532.793,Z 207.162,A -85,B 0,C 180,E1 -4395.27,E2 -4395.27} C_VEL
LIN {X 0,Y 532.447,Z 300.385,A -85,B 0,C 180,E1 -4396.548,E2 -4396.548} C_VEL
LIN {X 0,Y 532.302,Z 310.28,A -85,B 0,C 180,E1 -4396.763,E2 -4396.763} C_VEL
LIN {X 0,Y 532.137,Z 320.258,A -85,B 0,C 180,E1 -4397.074,E2 -4397.074} C_VEL
LIN {X 0,Y 531.938,Z 329.616,A -85,B 0,C 180,E1 -4397.457,E2 -4397.457} C_VEL
LIN {X 0,Y 531.74,Z 339.61,A -85,B 0,C 180,E1 -4397.976,E2 -4397.976} C_VEL
LIN {X 0,Y 531.536,Z 348.761,A -85,B 0,C 180,E1 -4398.561,E2 -4398.561} C_VEL
LIN {X 0,Y 531.333,Z 357.493,A -85,B 0,C 180,E1 -4399.232,E2 -4399.232} C_VEL
LIN {X 0,Y 531.147,Z 364.89,A -85,B 0,C 180,E1 -4399.903,E2 -4399.903} C_VEL
LIN {X 0,Y 530.974,Z 372.111,A -85,B 0,C 180,E1 -4400.669,E2 -4400.669} C_VEL
LIN {X 0,Y 530.857,Z 378.314,A -85,B 0,C 180,E1 -4401.435,E2 -4401.435} C_VEL
LIN {X 0,Y 530.684,Z 384.849,A -85,B 0,C 180,E1 -4402.39,E2 -4402.39} C_VEL
LIN {X 0,Y 530.557,Z 390.876,A -85,B 0,C 180,E1 -4403.458,E2 -4403.458} C_VEL
LIN {X 0,Y 530.572,Z 394.839,A -85,B 0,C 180,E1 -4404.299,E2 -4404.299} C_VEL
LIN {X 0,Y 530.456,Z 399.157,A -85,B 0,C 180,E1 -4405.441,E2 -4405.441} C_VEL
LIN {X 0,Y 530.516,Z 401.522,A -85,B 0,C 180,E1 -4406.202,E2 -4406.202} C_VEL
LIN {X 0,Y 530.457,Z 403.315,A -85,B 0,C 180,E1 -4406.962,E2 -4406.962} C_VEL
LIN {X 0,Y 530.361,Z 405.752,A -85,B 0,C 180,E1 -4408.481,E2 -4408.481} C_VEL
LIN {X 0,Y 530.347,Z 406.338,A -85,B 0,C 180,E1 -4409.241,E2 -4409.241} C_VEL
LIN {X 0,Y 530.347,Z 406.338,A -85,B 0,C 180,E1 -4410.759,E2 -4410.759} C_VEL
LIN {X 0,Y 530.361,Z 405.752,A -85,B 0,C 180,E1 -4411.519,E2 -4411.519} C_VEL
LIN {X 0,Y 530.457,Z 403.315,A -85,B 0,C 180,E1 -4413.038,E2 -4413.038} C_VEL
LIN {X 0,Y 530.523,Z 400.374,A -85,B 0,C 180,E1 -4414.178,E2 -4414.178} C_VEL
LIN {X 0,Y 530.52,Z 396.39,A -85,B 0,C 180,E1 -4415.321,E2 -4415.321} C_VEL
LIN {X 0,Y 530.533,Z 392.122,A -85,B 0,C 180,E1 -4416.294,E2 -4416.294} C_VEL
LIN {X 0,Y 530.666,Z 387.161,A -85,B 0,C 180,E1 -4417.228,E2 -4417.228} C_VEL
LIN {X 0,Y 530.774,Z 381.065,A -85,B 0,C 180,E1 -4418.183,E2 -4418.183} C_VEL
LIN {X 0,Y 530.912,Z 373.737,A -85,B 0,C 180,E1 -4419.14,E2 -4419.14} C_VEL
LIN {X 0,Y 531.072,Z 366.809,A -85,B 0,C 180,E1 -4419.906,E2 -4419.906} C_VEL
LIN {X 0,Y 531.317,Z 358.628,A -85,B 0,C 180,E1 -4420.672,E2 -4420.672} C_VEL
LIN {X 0,Y 531.511,Z 350.114,A -85,B 0,C 180,E1 -4421.343,E2 -4421.343} C_VEL
LIN {X 0,Y 531.694,Z 340.886,A -85,B 0,C 180,E1 -4421.949,E2 -4421.949} C_VEL
LIN {X 0,Y 531.911,Z 331.631,A -85,B 0,C 180,E1 -4422.447,E2 -4422.447} C_VEL
LIN {X 0,Y 532.095,Z 322.835,A -85,B 0,C 180,E1 -4422.83,E2 -4422.83} C_VEL
LIN {X 0,Y 532.273,Z 312.904,A -85,B 0,C 180,E1 -4423.165,E2 -4423.165} C_VEL
LIN {X 0,Y 532.37,Z 303.047,A -85,B 0,C 180,E1 -4423.406,E2 -4423.406} C_VEL
LIN {X 0,Y 532.564,Z 278.439,A -85,B 0,C 180,E1 -4423.765,E2 -4423.765} C_VEL
LIN {X 0,Y 532.651,Z 205.154,A -85,B 0,C 180,E1 -4424.761,E2 -4424.761} C_VEL
LIN {X 0,Y 531.148,Z 195.887,A -85,B 0,C 180,E1 -4424.943,E2 -4424.943} C_VEL
LIN {X 0,Y 531.086,Z 194.502,A -85,B 0,C 180,E1 -4425.127,E2 -4425.127} C_VEL
LIN {X 0,Y 531.366,Z 180.699,A -85,B 0,C 180,E1 -4427.768,E2 -4427.768} C_VEL
LIN {X 0,Y 531.648,Z 165.327,A -85,B 0,C 180,E1 -4430.708,E2 -4430.708} C_VEL
LIN {X 0,Y 531.997,Z 149.783,A -85,B 0,C 180,E1 -4433.761,E2 -4433.761} C_VEL
LIN {X 0,Y 531.893,Z 144.598,A -85,B 0,C 180,E1 -4434.809,E2 -4434.809} C_VEL
LIN {X 0,Y 531.045,Z 139.865,A -85,B 0,C 180,E1 -4435.862,E2 -4435.862} C_VEL
LIN {X 0,Y 530.977,Z 139.845,A -85,B 0,C 180,E1 -4438.456,E2 -4438.456} C_VEL
LIN {X 0,Y 530.959,Z 139.844,A -85,B 0,C 180,E1 -4441.079,E2 -4441.079} C_VEL
LIN {X 0,Y 530.988,Z 139.846,A -85,B 0,C 180,E1 -4443.772,E2 -4443.772} C_VEL
LIN {X 0,Y 530.956,Z 139.843,A -85,B 0,C 180,E1 -4446.558,E2 -4446.558} C_VEL
LIN {X 0,Y 530.99,Z 139.842,A -85,B 0,C 180,E1 -4449.443,E2 -4449.443} C_VEL
LIN {X 0,Y 530.977,Z 139.84,A -85,B 0,C 180,E1 -4452.456,E2 -4452.456} C_VEL
LIN {X 0,Y 530.977,Z 139.846,A -85,B 0,C 180,E1 -4455.621,E2 -4455.621} C_VEL
LIN {X 0,Y 530.992,Z 139.837,A -85,B 0,C 180,E1 -4458.564,E2 -4458.564} C_VEL
LIN {X 0,Y 530.956,Z 139.849,A -85,B 0,C 180,E1 -4461.529,E2 -4461.529} C_VEL
LIN {X 0,Y 530.955,Z 139.841,A -85,B 0,C 180,E1 -4464.38,E2 -4464.38} C_VEL
LIN {X 0,Y 530.969,Z 139.843,A -85,B 0,C 180,E1 -4467.133,E2 -4467.133} C_VEL
LIN {X 0,Y 530.968,Z 139.842,A -85,B 0,C 180,E1 -4469.803,E2 -4469.803} C_VEL
LIN {X 0,Y 531.011,Z 139.832,A -85,B 0,C 180,E1 -4472.467,E2 -4472.467} C_VEL
LIN {X 0,Y 531.003,Z 139.839,A -85,B 0,C 180,E1 -4474.942,E2 -4474.942} C_VEL
LIN {X 0,Y 530.969,Z 139.84,A -85,B 0,C 180,E1 -4478.246,E2 -4478.246} C_VEL
LIN {X 0,Y 530.994,Z 139.838,A -85,B 0,C 180,E1 -4480.677,E2 -4480.677} C_VEL
LIN {X 0,Y 530.983,Z 139.842,A -85,B 0,C 180,E1 -4483.071,E2 -4483.071} C_VEL
LIN {X 0,Y 531.017,Z 139.835,A -85,B 0,C 180,E1 -4485.435,E2 -4485.435} C_VEL
LIN {X 0,Y 531.034,Z 139.837,A -85,B 0,C 180,E1 -4488.549,E2 -4488.549} C_VEL
LIN {X 0,Y 531.052,Z 139.824,A -85,B 0,C 180,E1 -4491.629,E2 -4491.629} C_VEL
LIN {X 0,Y 531.118,Z 139.829,A -85,B 0,C 180,E1 -4494.685,E2 -4494.685} C_VEL
LIN {X 0,Y 531.135,Z 139.818,A -85,B 0,C 180,E1 -4497.725,E2 -4497.725} C_VEL
LIN {X 0,Y 531.15,Z 139.815,A -85,B 0,C 180,E1 -4500.758,E2 -4500.758} C_VEL
LIN {X 0,Y 531.102,Z 139.823,A -85,B 0,C 180,E1 -4503.034,E2 -4503.034} C_VEL
LIN {X 0,Y 531.08,Z 139.834,A -85,B 0,C 180,E1 -4506.077,E2 -4506.077} C_VEL
LIN {X 0,Y 531.026,Z 139.826,A -85,B 0,C 180,E1 -4509.138,E2 -4509.138} C_VEL
LIN {X 0,Y 531.036,Z 139.838,A -85,B 0,C 180,E1 -4512.225,E2 -4512.225} C_VEL
LIN {X 0,Y 530.991,Z 139.839,A -85,B 0,C 180,E1 -4515.349,E2 -4515.349} C_VEL
LIN {X 0,Y 530.989,Z 139.831,A -85,B 0,C 180,E1 -4518.521,E2 -4518.521} C_VEL
LIN {X 0,Y 530.995,Z 139.834,A -85,B 0,C 180,E1 -4520.938,E2 -4520.938} C_VEL
LIN {X 0,Y 530.975,Z 139.841,A -85,B 0,C 180,E1 -4524.224,E2 -4524.224} C_VEL
LIN {X 0,Y 531.007,Z 139.83,A -85,B 0,C 180,E1 -4526.743,E2 -4526.743} C_VEL
LIN {X 0,Y 530.977,Z 139.841,A -85,B 0,C 180,E1 -4529.322,E2 -4529.322} C_VEL
LIN {X 0,Y 530.975,Z 139.841,A -85,B 0,C 180,E1 -4532.103,E2 -4532.103} C_VEL
LIN {X 0,Y 530.986,Z 139.834,A -85,B 0,C 180,E1 -4534.854,E2 -4534.854} C_VEL
LIN {X 0,Y 530.961,Z 139.849,A -85,B 0,C 180,E1 -4537.507,E2 -4537.507} C_VEL
LIN {X 0,Y 530.98,Z 139.836,A -85,B 0,C 180,E1 -4540.432,E2 -4540.432} C_VEL
LIN {X 0,Y 530.963,Z 139.846,A -85,B 0,C 180,E1 -4543.494,E2 -4543.494} C_VEL
LIN {X 0,Y 530.96,Z 139.846,A -85,B 0,C 180,E1 -4543.558,E2 -4543.558} C_VEL
LIN {X 0,Y 530.286,Z 139.926,A -85,B 0,C 180,E1 -4544.192,E2 -4544.192} C_VEL
LIN {X 0,Y 527.437,Z 140.285,A -85,B 0,C 180,E1 -4545.22,E2 -4545.22} C_VEL
LIN {X 0,Y 525.033,Z 140.586,A -85,B 0,C 180,E1 -4546.049,E2 -4546.049} C_VEL
LIN {X 0,Y 524,Z 140.71,A -85,B 0,C 180,E1 -4546.688,E2 -4546.688} C_VEL
LIN {X 0,Y 523.914,Z 140.717,A -85,B 0,C 180,E1 -4546.905,E2 -4546.905} C_VEL
LIN {X 0,Y 523.932,Z 140.715,A -85,B 0,C 180,E1 -4549.87,E2 -4549.87} C_VEL
LIN {X 0,Y 523.907,Z 140.728,A -85,B 0,C 180,E1 -4552.868,E2 -4552.868} C_VEL
LIN {X 0,Y 523.939,Z 140.711,A -85,B 0,C 180,E1 -4555.711,E2 -4555.711} C_VEL
LIN {X 0,Y 523.929,Z 140.722,A -85,B 0,C 180,E1 -4558.457,E2 -4558.457} C_VEL
LIN {X 0,Y 523.94,Z 140.719,A -85,B 0,C 180,E1 -4561.126,E2 -4561.126} C_VEL
LIN {X 0,Y 523.98,Z 140.713,A -85,B 0,C 180,E1 -4563.98,E2 -4563.98} C_VEL
LIN {X 0,Y 523.933,Z 140.722,A -85,B 0,C 180,E1 -4566.271,E2 -4566.271} C_VEL
LIN {X 0,Y 523.943,Z 140.723,A -85,B 0,C 180,E1 -4568.767,E2 -4568.767} C_VEL
LIN {X 0,Y 523.948,Z 140.718,A -85,B 0,C 180,E1 -4571.221,E2 -4571.221} C_VEL
LIN {X 0,Y 523.934,Z 140.719,A -85,B 0,C 180,E1 -4573.639,E2 -4573.639} C_VEL
LIN {X 0,Y 523.937,Z 140.722,A -85,B 0,C 180,E1 -4576.028,E2 -4576.028} C_VEL
LIN {X 0,Y 524.009,Z 140.716,A -85,B 0,C 180,E1 -4578.394,E2 -4578.394} C_VEL
LIN {X 0,Y 524.002,Z 140.711,A -85,B 0,C 180,E1 -4581.516,E2 -4581.516} C_VEL
LIN {X 0,Y 524.081,Z 140.704,A -85,B 0,C 180,E1 -4584.614,E2 -4584.614} C_VEL
LIN {X 0,Y 524.111,Z 140.701,A -85,B 0,C 180,E1 -4587.695,E2 -4587.695} C_VEL
LIN {X 0,Y 524.121,Z 140.696,A -85,B 0,C 180,E1 -4590.768,E2 -4590.768} C_VEL
LIN {X 0,Y 524.069,Z 140.702,A -85,B 0,C 180,E1 -4593.075,E2 -4593.075} C_VEL
LIN {X 0,Y 524.045,Z 140.709,A -85,B 0,C 180,E1 -4596.159,E2 -4596.159} C_VEL
LIN {X 0,Y 523.997,Z 140.714,A -85,B 0,C 180,E1 -4599.262,E2 -4599.262} C_VEL
LIN {X 0,Y 524,Z 140.717,A -85,B 0,C 180,E1 -4601.74,E2 -4601.74} C_VEL
LIN {X 0,Y 523.989,Z 140.714,A -85,B 0,C 180,E1 -4605.052,E2 -4605.052} C_VEL
LIN {X 0,Y 523.96,Z 140.718,A -85,B 0,C 180,E1 -4607.969,E2 -4607.969} C_VEL
LIN {X 0,Y 523.968,Z 140.714,A -85,B 0,C 180,E1 -4610.41,E2 -4610.41} C_VEL
LIN {X 0,Y 523.913,Z 140.723,A -85,B 0,C 180,E1 -4612.893,E2 -4612.893} C_VEL
LIN {X 0,Y 523.949,Z 140.723,A -85,B 0,C 180,E1 -4615.419,E2 -4615.419} C_VEL
LIN {X 0,Y 523.966,Z 140.713,A -85,B 0,C 180,E1 -4617.999,E2 -4617.999} C_VEL
LIN {X 0,Y 523.949,Z 140.717,A -85,B 0,C 180,E1 -4620.856,E2 -4620.856} C_VEL
LIN {X 0,Y 523.956,Z 140.709,A -85,B 0,C 180,E1 -4623.735,E2 -4623.735} C_VEL
LIN {X 0,Y 523.915,Z 140.718,A -85,B 0,C 180,E1 -4626.404,E2 -4626.404} C_VEL
LIN {X 0,Y 523.92,Z 140.723,A -85,B 0,C 180,E1 -4629.084,E2 -4629.084} C_VEL
LIN {X 0,Y 523.951,Z 140.701,A -85,B 0,C 180,E1 -4632.118,E2 -4632.118} C_VEL
LIN {X 0,Y 523.951,Z 140.717,A -85,B 0,C 180,E1 -4635.309,E2 -4635.309} C_VEL
LIN {X 0,Y 523.957,Z 140.718,A -85,B 0,C 180,E1 -4638.689,E2 -4638.689} C_VEL
LIN {X 0,Y 523.912,Z 140.721,A -85,B 0,C 180,E1 -4641.898,E2 -4641.898} C_VEL
LIN {X 0,Y 523.934,Z 140.714,A -85,B 0,C 180,E1 -4644.909,E2 -4644.909} C_VEL
LIN {X 0,Y 523.938,Z 140.716,A -85,B 0,C 180,E1 -4647.678,E2 -4647.678} C_VEL
LIN {X 0,Y 523.949,Z 140.717,A -85,B 0,C 180,E1 -4650.676,E2 -4650.676} C_VEL
LIN {X 0,Y 523.973,Z 140.708,A -85,B 0,C 180,E1 -4653.729,E2 -4653.729} C_VEL
LIN {X 0,Y 523.932,Z 140.726,A -85,B 0,C 180,E1 -4656.271,E2 -4656.271} C_VEL
LIN {X 0,Y 523.941,Z 140.714,A -85,B 0,C 180,E1 -4658.767,E2 -4658.767} C_VEL
LIN {X 0,Y 523.949,Z 140.706,A -85,B 0,C 180,E1 -4661.221,E2 -4661.221} C_VEL
LIN {X 0,Y 523.933,Z 140.718,A -85,B 0,C 180,E1 -4663.639,E2 -4663.639} C_VEL
LIN {X 0,Y 523.937,Z 140.724,A -85,B 0,C 180,E1 -4666.028,E2 -4666.028} C_VEL
LIN {X 0,Y 524.008,Z 140.704,A -85,B 0,C 180,E1 -4668.394,E2 -4668.394} C_VEL
LIN {X 0,Y 524,Z 140.705,A -85,B 0,C 180,E1 -4671.516,E2 -4671.516} C_VEL
LIN {X 0,Y 524.079,Z 140.699,A -85,B 0,C 180,E1 -4674.614,E2 -4674.614} C_VEL
LIN {X 0,Y 524.107,Z 140.698,A -85,B 0,C 180,E1 -4677.695,E2 -4677.695} C_VEL
LIN {X 0,Y 524.12,Z 140.686,A -85,B 0,C 180,E1 -4680.769,E2 -4680.769} C_VEL
LIN {X 0,Y 524.069,Z 140.7,A -85,B 0,C 180,E1 -4683.075,E2 -4683.075} C_VEL
LIN {X 0,Y 524.043,Z 140.703,A -85,B 0,C 180,E1 -4686.159,E2 -4686.159} C_VEL
LIN {X 0,Y 523.994,Z 140.708,A -85,B 0,C 180,E1 -4689.262,E2 -4689.262} C_VEL
LIN {X 0,Y 523.999,Z 140.709,A -85,B 0,C 180,E1 -4691.74,E2 -4691.74} C_VEL
LIN {X 0,Y 523.99,Z 140.716,A -85,B 0,C 180,E1 -4695.053,E2 -4695.053} C_VEL
LIN {X 0,Y 523.962,Z 140.705,A -85,B 0,C 180,E1 -4697.969,E2 -4697.969} C_VEL
LIN {X 0,Y 523.97,Z 140.708,A -85,B 0,C 180,E1 -4700.411,E2 -4700.411} C_VEL
LIN {X 0,Y 523.909,Z 140.726,A -85,B 0,C 180,E1 -4702.894,E2 -4702.894} C_VEL
LIN {X 0,Y 523.951,Z 140.712,A -85,B 0,C 180,E1 -4705.419,E2 -4705.419} C_VEL
LIN {X 0,Y 523.966,Z 140.708,A -85,B 0,C 180,E1 -4708,E2 -4708} C_VEL
LIN {X 0,Y 523.943,Z 140.724,A -85,B 0,C 180,E1 -4710.855,E2 -4710.855} C_VEL
LIN {X 0,Y 523.959,Z 140.709,A -85,B 0,C 180,E1 -4713.735,E2 -4713.735} C_VEL
LIN {X 0,Y 523.902,Z 140.724,A -85,B 0,C 180,E1 -4716.402,E2 -4716.402} C_VEL
LIN {X 0,Y 523.919,Z 140.718,A -85,B 0,C 180,E1 -4719.085,E2 -4719.085} C_VEL
LIN {X 0,Y 523.95,Z 140.718,A -85,B 0,C 180,E1 -4722.12,E2 -4722.12} C_VEL
LIN {X 0,Y 523.943,Z 140.715,A -85,B 0,C 180,E1 -4725.311,E2 -4725.311} C_VEL
LIN {X 0,Y 523.956,Z 140.712,A -85,B 0,C 180,E1 -4728.69,E2 -4728.69} C_VEL
LIN {X 0,Y 523.92,Z 140.718,A -85,B 0,C 180,E1 -4731.081,E2 -4731.081} C_VEL
LIN {X 0,Y 523.901,Z 140.725,A -85,B 0,C 180,E1 -4733.826,E2 -4733.826} C_VEL
LIN {X 0,Y 523.942,Z 140.718,A -85,B 0,C 180,E1 -4736.636,E2 -4736.636} C_VEL
LIN {X 0,Y 523.958,Z 140.718,A -85,B 0,C 180,E1 -4739.356,E2 -4739.356} C_VEL
LIN {X 0,Y 523.978,Z 140.716,A -85,B 0,C 180,E1 -4742.282,E2 -4742.282} C_VEL
LIN {X 0,Y 524.001,Z 140.858,A -85,B 0,C 180,E1 -4744.021,E2 -4744.021} C_VEL
LIN {X 0,Y 525.087,Z 147.777,A -85,B 0,C 180,E1 -4745.526,E2 -4745.526} C_VEL
LIN {X 0,Y 524.72,Z 162.054,A -85,B 0,C 180,E1 -4748.388,E2 -4748.388} C_VEL
LIN {X 0,Y 524.411,Z 175.65,A -85,B 0,C 180,E1 -4751.035,E2 -4751.035} C_VEL
LIN {X 0,Y 524.138,Z 190.148,A -85,B 0,C 180,E1 -4753.846,E2 -4753.846} C_VEL
LIN {X 0,Y 524.055,Z 195.318,A -85,B 0,C 180,E1 -4754.826,E2 -4754.826} C_VEL
LIN {X 0,Y 525.213,Z 202.515,A -85,B 0,C 180,E1 -4754.991,E2 -4754.991} C_VEL
LIN {X 0,Y 525.934,Z 208.105,A -85,B 0,C 180,E1 -4755.089,E2 -4755.089} C_VEL
LIN {X 0,Y 525.544,Z 300.193,A -85,B 0,C 180,E1 -4756.368,E2 -4756.368} C_VEL
LIN {X 0,Y 525.391,Z 310.089,A -85,B 0,C 180,E1 -4756.585,E2 -4756.585} C_VEL
LIN {X 0,Y 525.224,Z 320.067,A -85,B 0,C 180,E1 -4756.901,E2 -4756.901} C_VEL
LIN {X 0,Y 525.006,Z 329.424,A -85,B 0,C 180,E1 -4757.289,E2 -4757.289} C_VEL
LIN {X 0,Y 524.762,Z 339.52,A -85,B 0,C 180,E1 -4757.82,E2 -4757.82} C_VEL
LIN {X 0,Y 524.55,Z 348.569,A -85,B 0,C 180,E1 -4758.406,E2 -4758.406} C_VEL
LIN {X 0,Y 524.333,Z 357.3,A -85,B 0,C 180,E1 -4759.087,E2 -4759.087} C_VEL
LIN {X 0,Y 524.14,Z 364.698,A -85,B 0,C 180,E1 -4759.766,E2 -4759.766} C_VEL
LIN {X 0,Y 523.956,Z 371.919,A -85,B 0,C 180,E1 -4760.543,E2 -4760.543} C_VEL
LIN {X 0,Y 523.788,Z 378.121,A -85,B 0,C 180,E1 -4761.318,E2 -4761.318} C_VEL
LIN {X 0,Y 523.629,Z 384.657,A -85,B 0,C 180,E1 -4762.287,E2 -4762.287} C_VEL
LIN {X 0,Y 523.512,Z 389.157,A -85,B 0,C 180,E1 -4763.061,E2 -4763.061} C_VEL
LIN {X 0,Y 523.487,Z 394.647,A -85,B 0,C 180,E1 -4764.221,E2 -4764.221} C_VEL
LIN {X 0,Y 523.361,Z 398.964,A -85,B 0,C 180,E1 -4765.379,E2 -4765.379} C_VEL
LIN {X 0,Y 523.444,Z 401.33,A -85,B 0,C 180,E1 -4766.151,E2 -4766.151} C_VEL
LIN {X 0,Y 523.368,Z 403.124,A -85,B 0,C 180,E1 -4766.921,E2 -4766.921} C_VEL
LIN {X 0,Y 523.275,Z 405.56,A -85,B 0,C 180,E1 -4768.461,E2 -4768.461} C_VEL
LIN {X 0,Y 523.253,Z 406.147,A -85,B 0,C 180,E1 -4769.23,E2 -4769.23} C_VEL
LIN {X 0,Y 523.253,Z 406.147,A -85,B 0,C 180,E1 -4770.77,E2 -4770.77} C_VEL
LIN {X 0,Y 523.275,Z 405.56,A -85,B 0,C 180,E1 -4771.539,E2 -4771.539} C_VEL
LIN {X 0,Y 523.368,Z 403.123,A -85,B 0,C 180,E1 -4773.079,E2 -4773.079} C_VEL
LIN {X 0,Y 523.425,Z 400.182,A -85,B 0,C 180,E1 -4774.235,E2 -4774.235} C_VEL
LIN {X 0,Y 523.455,Z 396.199,A -85,B 0,C 180,E1 -4775.393,E2 -4775.393} C_VEL
LIN {X 0,Y 523.471,Z 391.181,A -85,B 0,C 180,E1 -4776.531,E2 -4776.531} C_VEL
LIN {X 0,Y 523.595,Z 385.812,A -85,B 0,C 180,E1 -4777.52,E2 -4777.52} C_VEL
LIN {X 0,Y 523.754,Z 379.497,A -85,B 0,C 180,E1 -4778.488,E2 -4778.488} C_VEL
LIN {X 0,Y 523.887,Z 373.545,A -85,B 0,C 180,E1 -4779.264,E2 -4779.264} C_VEL
LIN {X 0,Y 524.041,Z 366.616,A -85,B 0,C 180,E1 -4780.04,E2 -4780.04} C_VEL
LIN {X 0,Y 524.315,Z 358.436,A -85,B 0,C 180,E1 -4780.816,E2 -4780.816} C_VEL
LIN {X 0,Y 524.523,Z 349.921,A -85,B 0,C 180,E1 -4781.496,E2 -4781.496} C_VEL
LIN {X 0,Y 524.742,Z 340.532,A -85,B 0,C 180,E1 -4782.12,E2 -4782.12} C_VEL
LIN {X 0,Y 524.973,Z 330.431,A -85,B 0,C 180,E1 -4782.663,E2 -4782.663} C_VEL
LIN {X 0,Y 525.188,Z 321.354,A -85,B 0,C 180,E1 -4783.051,E2 -4783.051} C_VEL
LIN {X 0,Y 525.393,Z 311.839,A -85,B 0,C 180,E1 -4783.366,E2 -4783.366} C_VEL
LIN {X 0,Y 525.507,Z 301.524,A -85,B 0,C 180,E1 -4783.609,E2 -4783.609} C_VEL
LIN {X 0,Y 525.83,Z 229.916,A -85,B 0,C 180,E1 -4784.612,E2 -4784.612} C_VEL
LIN {X 0,Y 525.748,Z 205.696,A -85,B 0,C 180,E1 -4784.949,E2 -4784.949} C_VEL
LIN {X 0,Y 524.066,Z 195.516,A -85,B 0,C 180,E1 -4785.159,E2 -4785.159} C_VEL
LIN {X 0,Y 524.072,Z 193.229,A -85,B 0,C 180,E1 -4785.557,E2 -4785.557} C_VEL
LIN {X 0,Y 524.375,Z 177.74,A -85,B 0,C 180,E1 -4788.561,E2 -4788.561} C_VEL
LIN {X 0,Y 524.653,Z 164.147,A -85,B 0,C 180,E1 -4791.203,E2 -4791.203} C_VEL
LIN {X 0,Y 525.091,Z 149.759,A -85,B 0,C 180,E1 -4794.075,E2 -4794.075} C_VEL
LIN {X 0,Y 524.878,Z 145.552,A -85,B 0,C 180,E1 -4794.947,E2 -4794.947} C_VEL
LIN {X 0,Y 523.973,Z 140.741,A -85,B 0,C 180,E1 -4796.043,E2 -4796.043} C_VEL
LIN {X 0,Y 523.932,Z 140.72,A -85,B 0,C 180,E1 -4798.875,E2 -4798.875} C_VEL
LIN {X 0,Y 523.923,Z 140.725,A -85,B 0,C 180,E1 -4801.544,E2 -4801.544} C_VEL
LIN {X 0,Y 523.934,Z 140.719,A -85,B 0,C 180,E1 -4804.29,E2 -4804.29} C_VEL
LIN {X 0,Y 523.908,Z 140.721,A -85,B 0,C 180,E1 -4807.132,E2 -4807.132} C_VEL
LIN {X 0,Y 523.938,Z 140.713,A -85,B 0,C 180,E1 -4810.129,E2 -4810.129} C_VEL
LIN {X 0,Y 523.935,Z 140.717,A -85,B 0,C 180,E1 -4812.458,E2 -4812.458} C_VEL
LIN {X 0,Y 523.943,Z 140.72,A -85,B 0,C 180,E1 -4815.31,E2 -4815.31} C_VEL
LIN {X 0,Y 523.955,Z 140.715,A -85,B 0,C 180,E1 -4818.689,E2 -4818.689} C_VEL
LIN {X 0,Y 523.916,Z 140.72,A -85,B 0,C 180,E1 -4821.08,E2 -4821.08} C_VEL
LIN {X 0,Y 523.899,Z 140.722,A -85,B 0,C 180,E1 -4823.825,E2 -4823.825} C_VEL
LIN {X 0,Y 523.941,Z 140.712,A -85,B 0,C 180,E1 -4826.635,E2 -4826.635} C_VEL
LIN {X 0,Y 523.955,Z 140.72,A -85,B 0,C 180,E1 -4829.355,E2 -4829.355} C_VEL
LIN {X 0,Y 523.975,Z 140.707,A -85,B 0,C 180,E1 -4832.281,E2 -4832.281} C_VEL
LIN {X 0,Y 523.951,Z 140.712,A -85,B 0,C 180,E1 -4834.581,E2 -4834.581} C_VEL
LIN {X 0,Y 523.909,Z 140.726,A -85,B 0,C 180,E1 -4837.106,E2 -4837.106} C_VEL
LIN {X 0,Y 523.976,Z 140.706,A -85,B 0,C 180,E1 -4839.865,E2 -4839.865} C_VEL
LIN {X 0,Y 523.964,Z 140.714,A -85,B 0,C 180,E1 -4842.837,E2 -4842.837} C_VEL
LIN {X 0,Y 523.974,Z 140.714,A -85,B 0,C 180,E1 -4845.235,E2 -4845.235} C_VEL
LIN {X 0,Y 524.009,Z 140.709,A -85,B 0,C 180,E1 -4848.394,E2 -4848.394} C_VEL
LIN {X 0,Y 524,Z 140.702,A -85,B 0,C 180,E1 -4851.516,E2 -4851.516} C_VEL
LIN {X 0,Y 524.079,Z 140.707,A -85,B 0,C 180,E1 -4854.613,E2 -4854.613} C_VEL
LIN {X 0,Y 524.108,Z 140.693,A -85,B 0,C 180,E1 -4857.694,E2 -4857.694} C_VEL
LIN {X 0,Y 524.12,Z 140.69,A -85,B 0,C 180,E1 -4860.768,E2 -4860.768} C_VEL
LIN {X 0,Y 524.069,Z 140.699,A -85,B 0,C 180,E1 -4863.074,E2 -4863.074} C_VEL
LIN {X 0,Y 524.042,Z 140.712,A -85,B 0,C 180,E1 -4866.159,E2 -4866.159} C_VEL
LIN {X 0,Y 523.994,Z 140.701,A -85,B 0,C 180,E1 -4869.261,E2 -4869.261} C_VEL
LIN {X 0,Y 523.998,Z 140.707,A -85,B 0,C 180,E1 -4871.739,E2 -4871.739} C_VEL
LIN {X 0,Y 523.988,Z 140.71,A -85,B 0,C 180,E1 -4875.052,E2 -4875.052} C_VEL
LIN {X 0,Y 523.96,Z 140.713,A -85,B 0,C 180,E1 -4877.969,E2 -4877.969} C_VEL
LIN {X 0,Y 523.967,Z 140.711,A -85,B 0,C 180,E1 -4880.41,E2 -4880.41} C_VEL
LIN {X 0,Y 523.912,Z 140.72,A -85,B 0,C 180,E1 -4882.893,E2 -4882.893} C_VEL
LIN {X 0,Y 523.951,Z 140.719,A -85,B 0,C 180,E1 -4885.418,E2 -4885.418} C_VEL
LIN {X 0,Y 523.966,Z 140.714,A -85,B 0,C 180,E1 -4887.999,E2 -4887.999} C_VEL
LIN {X 0,Y 523.942,Z 140.717,A -85,B 0,C 180,E1 -4890.855,E2 -4890.855} C_VEL
LIN {X 0,Y 523.958,Z 140.713,A -85,B 0,C 180,E1 -4893.735,E2 -4893.735} C_VEL
LIN {X 0,Y 523.917,Z 140.718,A -85,B 0,C 180,E1 -4896.404,E2 -4896.404} C_VEL
LIN {X 0,Y 523.918,Z 140.724,A -85,B 0,C 180,E1 -4899.084,E2 -4899.084} C_VEL
LIN {X 0,Y 523.953,Z 140.714,A -85,B 0,C 180,E1 -4902.118,E2 -4902.118} C_VEL
LIN {X 0,Y 523.951,Z 140.716,A -85,B 0,C 180,E1 -4905.309,E2 -4905.309} C_VEL
LIN {X 0,Y 523.914,Z 140.717,A -85,B 0,C 180,E1 -4906.905,E2 -4906.905} C_VEL
LIN {X 0,Y 523.247,Z 140.791,A -85,B 0,C 180,E1 -4907.546,E2 -4907.546} C_VEL
LIN {X 0,Y 520.404,Z 141.144,A -85,B 0,C 180,E1 -4908.588,E2 -4908.588} C_VEL
LIN {X 0,Y 518,Z 141.457,A -85,B 0,C 180,E1 -4909.427,E2 -4909.427} C_VEL
LIN {X 0,Y 516.964,Z 141.583,A -85,B 0,C 180,E1 -4910.074,E2 -4910.074} C_VEL
LIN {X 0,Y 516.877,Z 141.593,A -85,B 0,C 180,E1 -4910.294,E2 -4910.294} C_VEL
LIN {X 0,Y 516.88,Z 141.596,A -85,B 0,C 180,E1 -4913.342,E2 -4913.342} C_VEL
LIN {X 0,Y 516.908,Z 141.586,A -85,B 0,C 180,E1 -4916.121,E2 -4916.121} C_VEL
LIN {X 0,Y 516.89,Z 141.599,A -85,B 0,C 180,E1 -4918.935,E2 -4918.935} C_VEL
LIN {X 0,Y 516.917,Z 141.59,A -85,B 0,C 180,E1 -4921.585,E2 -4921.585} C_VEL
LIN {X 0,Y 516.928,Z 141.594,A -85,B 0,C 180,E1 -4924.211,E2 -4924.211} C_VEL
LIN {X 0,Y 516.869,Z 141.605,A -85,B 0,C 180,E1 -4926.777,E2 -4926.777} C_VEL
LIN {X 0,Y 516.936,Z 141.591,A -85,B 0,C 180,E1 -4929.732,E2 -4929.732} C_VEL
LIN {X 0,Y 516.925,Z 141.598,A -85,B 0,C 180,E1 -4932.596,E2 -4932.596} C_VEL
LIN {X 0,Y 516.939,Z 141.592,A -85,B 0,C 180,E1 -4935.03,E2 -4935.03} C_VEL
LIN {X 0,Y 516.962,Z 141.594,A -85,B 0,C 180,E1 -4938.234,E2 -4938.234} C_VEL
LIN {X 0,Y 516.967,Z 141.588,A -85,B 0,C 180,E1 -4941.4,E2 -4941.4} C_VEL
LIN {X 0,Y 517.009,Z 141.585,A -85,B 0,C 180,E1 -4943.757,E2 -4943.757} C_VEL
LIN {X 0,Y 517.083,Z 141.576,A -85,B 0,C 180,E1 -4947.663,E2 -4947.663} C_VEL
LIN {X 0,Y 517.091,Z 141.572,A -85,B 0,C 180,E1 -4950.779,E2 -4950.779} C_VEL
LIN {X 0,Y 517.01,Z 141.582,A -85,B 0,C 180,E1 -4953.117,E2 -4953.117} C_VEL
LIN {X 0,Y 517.009,Z 141.585,A -85,B 0,C 180,E1 -4956.243,E2 -4956.243} C_VEL
LIN {X 0,Y 516.952,Z 141.593,A -85,B 0,C 180,E1 -4959.389,E2 -4959.389} C_VEL
LIN {X 0,Y 516.949,Z 141.595,A -85,B 0,C 180,E1 -4961.808,E2 -4961.808} C_VEL
LIN {X 0,Y 516.941,Z 141.593,A -85,B 0,C 180,E1 -4965.146,E2 -4965.146} C_VEL
LIN {X 0,Y 516.922,Z 141.593,A -85,B 0,C 180,E1 -4968.222,E2 -4968.222} C_VEL
LIN {X 0,Y 516.909,Z 141.594,A -85,B 0,C 180,E1 -4970.701,E2 -4970.701} C_VEL
LIN {X 0,Y 516.908,Z 141.594,A -85,B 0,C 180,E1 -4974.072,E2 -4974.072} C_VEL
LIN {X 0,Y 516.923,Z 141.593,A -85,B 0,C 180,E1 -4976.658,E2 -4976.658} C_VEL
LIN {X 0,Y 516.921,Z 141.592,A -85,B 0,C 180,E1 -4979.527,E2 -4979.527} C_VEL
LIN {X 0,Y 516.896,Z 141.596,A -85,B 0,C 180,E1 -4982.544,E2 -4982.544} C_VEL
LIN {X 0,Y 516.875,Z 141.597,A -85,B 0,C 180,E1 -4985.332,E2 -4985.332} C_VEL
LIN {X 0,Y 516.877,Z 141.597,A -85,B 0,C 180,E1 -4987.943,E2 -4987.943} C_VEL
LIN {X 0,Y 516.88,Z 141.593,A -85,B 0,C 180,E1 -4990.741,E2 -4990.741} C_VEL
LIN {X 0,Y 516.879,Z 141.588,A -85,B 0,C 180,E1 -4992.831,E2 -4992.831} C_VEL
LIN {X 0,Y 516.917,Z 141.597,A -85,B 0,C 180,E1 -4995.01,E2 -4995.01} C_VEL
LIN {X 0,Y 516.912,Z 141.595,A -85,B 0,C 180,E1 -4998.398,E2 -4998.398} C_VEL
LIN {X 0,Y 516.877,Z 141.597,A -85,B 0,C 180,E1 -5001.284,E2 -5001.284} C_VEL
LIN {X 0,Y 516.886,Z 141.598,A -85,B 0,C 180,E1 -5004.221,E2 -5004.221} C_VEL
LIN {X 0,Y 516.894,Z 141.595,A -85,B 0,C 180,E1 -5007.054,E2 -5007.054} C_VEL
LIN {X 0,Y 516.887,Z 141.596,A -85,B 0,C 180,E1 -5009.797,E2 -5009.797} C_VEL
LIN {X 0,Y 516.925,Z 141.589,A -85,B 0,C 180,E1 -5012.468,E2 -5012.468} C_VEL
LIN {X 0,Y 516.907,Z 141.592,A -85,B 0,C 180,E1 -5015.072,E2 -5015.072} C_VEL
LIN {X 0,Y 516.881,Z 141.597,A -85,B 0,C 180,E1 -5018.463,E2 -5018.463} C_VEL
LIN {X 0,Y 516.9,Z 141.584,A -85,B 0,C 180,E1 -5020.955,E2 -5020.955} C_VEL
LIN {X 0,Y 516.909,Z 141.59,A -85,B 0,C 180,E1 -5023.411,E2 -5023.411} C_VEL
LIN {X 0,Y 516.892,Z 141.601,A -85,B 0,C 180,E1 -5025.834,E2 -5025.834} C_VEL
LIN {X 0,Y 516.961,Z 141.583,A -85,B 0,C 180,E1 -5028.234,E2 -5028.234} C_VEL
LIN {X 0,Y 516.965,Z 141.579,A -85,B 0,C 180,E1 -5031.4,E2 -5031.4} C_VEL
LIN {X 0,Y 517.006,Z 141.586,A -85,B 0,C 180,E1 -5033.757,E2 -5033.757} C_VEL
LIN {X 0,Y 517.079,Z 141.573,A -85,B 0,C 180,E1 -5037.664,E2 -5037.664} C_VEL
LIN {X 0,Y 517.09,Z 141.561,A -85,B 0,C 180,E1 -5040.779,E2 -5040.779} C_VEL
LIN {X 0,Y 517.01,Z 141.58,A -85,B 0,C 180,E1 -5043.117,E2 -5043.117} C_VEL
LIN {X 0,Y 517.007,Z 141.579,A -85,B 0,C 180,E1 -5046.244,E2 -5046.244} C_VEL
LIN {X 0,Y 516.948,Z 141.583,A -85,B 0,C 180,E1 -5049.39,E2 -5049.39} C_VEL
LIN {X 0,Y 516.949,Z 141.586,A -85,B 0,C 180,E1 -5051.808,E2 -5051.808} C_VEL
LIN {X 0,Y 516.941,Z 141.595,A -85,B 0,C 180,E1 -5055.147,E2 -5055.147} C_VEL
LIN {X 0,Y 516.923,Z 141.581,A -85,B 0,C 180,E1 -5058.223,E2 -5058.223} C_VEL
LIN {X 0,Y 516.91,Z 141.59,A -85,B 0,C 180,E1 -5060.702,E2 -5060.702} C_VEL
LIN {X 0,Y 516.901,Z 141.592,A -85,B 0,C 180,E1 -5064.073,E2 -5064.073} C_VEL
LIN {X 0,Y 516.922,Z 141.59,A -85,B 0,C 180,E1 -5066.658,E2 -5066.658} C_VEL
LIN {X 0,Y 516.91,Z 141.592,A -85,B 0,C 180,E1 -5069.524,E2 -5069.524} C_VEL
LIN {X 0,Y 516.896,Z 141.599,A -85,B 0,C 180,E1 -5072.544,E2 -5072.544} C_VEL
LIN {X 0,Y 516.867,Z 141.596,A -85,B 0,C 180,E1 -5075.331,E2 -5075.331} C_VEL
LIN {X 0,Y 516.879,Z 141.597,A -85,B 0,C 180,E1 -5077.944,E2 -5077.944} C_VEL
LIN {X 0,Y 516.882,Z 141.601,A -85,B 0,C 180,E1 -5080.742,E2 -5080.742} C_VEL
LIN {X 0,Y 516.882,Z 141.599,A -85,B 0,C 180,E1 -5082.832,E2 -5082.832} C_VEL
LIN {X 0,Y 516.895,Z 141.595,A -85,B 0,C 180,E1 -5085.007,E2 -5085.007} C_VEL
LIN {X 0,Y 516.913,Z 141.593,A -85,B 0,C 180,E1 -5088.399,E2 -5088.399} C_VEL
LIN {X 0,Y 516.883,Z 141.594,A -85,B 0,C 180,E1 -5091.285,E2 -5091.285} C_VEL
LIN {X 0,Y 516.872,Z 141.599,A -85,B 0,C 180,E1 -5094.22,E2 -5094.22} C_VEL
LIN {X 0,Y 516.896,Z 141.594,A -85,B 0,C 180,E1 -5097.054,E2 -5097.054} C_VEL
LIN {X 0,Y 516.894,Z 141.601,A -85,B 0,C 180,E1 -5099.797,E2 -5099.797} C_VEL
LIN {X 0,Y 516.928,Z 141.595,A -85,B 0,C 180,E1 -5102.468,E2 -5102.468} C_VEL
LIN {X 0,Y 516.95,Z 141.643,A -85,B 0,C 180,E1 -5103.803,E2 -5103.803} C_VEL
LIN {X 0,Y 518.111,Z 148.498,A -85,B 0,C 180,E1 -5105.345,E2 -5105.345} C_VEL
LIN {X 0,Y 517.794,Z 159.851,A -85,B 0,C 180,E1 -5107.664,E2 -5107.664} C_VEL
LIN {X 0,Y 517.533,Z 172.383,A -85,B 0,C 180,E1 -5110.154,E2 -5110.154} C_VEL
LIN {X 0,Y 517.185,Z 185.858,A -85,B 0,C 180,E1 -5112.809,E2 -5112.809} C_VEL
LIN {X 0,Y 517.048,Z 195.145,A -85,B 0,C 180,E1 -5114.618,E2 -5114.618} C_VEL
LIN {X 0,Y 518.365,Z 203.291,A -85,B 0,C 180,E1 -5114.802,E2 -5114.802} C_VEL
LIN {X 0,Y 519.056,Z 208.976,A -85,B 0,C 180,E1 -5114.902,E2 -5114.902} C_VEL
LIN {X 0,Y 518.647,Z 300.001,A -85,B 0,C 180,E1 -5116.183,E2 -5116.183} C_VEL
LIN {X 0,Y 518.478,Z 309.897,A -85,B 0,C 180,E1 -5116.403,E2 -5116.403} C_VEL
LIN {X 0,Y 518.303,Z 319.875,A -85,B 0,C 180,E1 -5116.723,E2 -5116.723} C_VEL
LIN {X 0,Y 518.063,Z 329.232,A -85,B 0,C 180,E1 -5117.115,E2 -5117.115} C_VEL
LIN {X 0,Y 517.85,Z 338.543,A -85,B 0,C 180,E1 -5117.607,E2 -5117.607} C_VEL
LIN {X 0,Y 517.64,Z 346.629,A -85,B 0,C 180,E1 -5118.121,E2 -5118.121} C_VEL
LIN {X 0,Y 517.32,Z 355.972,A -85,B 0,C 180,E1 -5118.838,E2 -5118.838} C_VEL
LIN {X 0,Y 517.106,Z 364.505,A -85,B 0,C 180,E1 -5119.626,E2 -5119.626} C_VEL
LIN {X 0,Y 516.935,Z 371.727,A -85,B 0,C 180,E1 -5120.413,E2 -5120.413} C_VEL
LIN {X 0,Y 516.71,Z 377.928,A -85,B 0,C 180,E1 -5121.198,E2 -5121.198} C_VEL
LIN {X 0,Y 516.547,Z 384.464,A -85,B 0,C 180,E1 -5122.18,E2 -5122.18} C_VEL
LIN {X 0,Y 516.439,Z 388.965,A -85,B 0,C 180,E1 -5122.965,E2 -5122.965} C_VEL
LIN {X 0,Y 516.401,Z 394.455,A -85,B 0,C 180,E1 -5124.142,E2 -5124.142} C_VEL
LIN {X 0,Y 516.272,Z 398.773,A -85,B 0,C 180,E1 -5125.315,E2 -5125.315} C_VEL
LIN {X 0,Y 516.352,Z 401.138,A -85,B 0,C 180,E1 -5126.098,E2 -5126.098} C_VEL
LIN {X 0,Y 516.283,Z 402.932,A -85,B 0,C 180,E1 -5126.879,E2 -5126.879} C_VEL
LIN {X 0,Y 516.192,Z 405.369,A -85,B 0,C 180,E1 -5128.44,E2 -5128.44} C_VEL
LIN {X 0,Y 516.162,Z 405.955,A -85,B 0,C 180,E1 -5129.22,E2 -5129.22} C_VEL
LIN {X 0,Y 516.162,Z 405.955,A -85,B 0,C 180,E1 -5130.78,E2 -5130.78} C_VEL
LIN {X 0,Y 516.192,Z 405.369,A -85,B 0,C 180,E1 -5131.56,E2 -5131.56} C_VEL
LIN {X 0,Y 516.283,Z 402.932,A -85,B 0,C 180,E1 -5133.121,E2 -5133.121} C_VEL
LIN {X 0,Y 516.313,Z 399.989,A -85,B 0,C 180,E1 -5134.293,E2 -5134.293} C_VEL
LIN {X 0,Y 516.367,Z 396.007,A -85,B 0,C 180,E1 -5135.467,E2 -5135.467} C_VEL
LIN {X 0,Y 516.386,Z 390.827,A -85,B 0,C 180,E1 -5136.654,E2 -5136.654} C_VEL
LIN {X 0,Y 516.533,Z 385.62,A -85,B 0,C 180,E1 -5137.623,E2 -5137.623} C_VEL
LIN {X 0,Y 516.709,Z 379.305,A -85,B 0,C 180,E1 -5138.605,E2 -5138.605} C_VEL
LIN {X 0,Y 516.851,Z 373.353,A -85,B 0,C 180,E1 -5139.391,E2 -5139.391} C_VEL
LIN {X 0,Y 517.02,Z 366.424,A -85,B 0,C 180,E1 -5140.178,E2 -5140.178} C_VEL
LIN {X 0,Y 517.31,Z 358.243,A -85,B 0,C 180,E1 -5140.964,E2 -5140.964} C_VEL
LIN {X 0,Y 517.536,Z 349.729,A -85,B 0,C 180,E1 -5141.654,E2 -5141.654} C_VEL
LIN {X 0,Y 517.751,Z 341.408,A -85,B 0,C 180,E1 -5142.221,E2 -5142.221} C_VEL
LIN {X 0,Y 518.016,Z 331.247,A -85,B 0,C 180,E1 -5142.786,E2 -5142.786} C_VEL
LIN {X 0,Y 518.238,Z 322.451,A -85,B 0,C 180,E1 -5143.179,E2 -5143.179} C_VEL
LIN {X 0,Y 518.469,Z 312.521,A -85,B 0,C 180,E1 -5143.522,E2 -5143.522} C_VEL
LIN {X 0,Y 518.577,Z 302.664,A -85,B 0,C 180,E1 -5143.769,E2 -5143.769} C_VEL
LIN {X 0,Y 518.797,Z 279.846,A -85,B 0,C 180,E1 -5144.113,E2 -5144.113} C_VEL
LIN {X 0,Y 518.878,Z 206.324,A -85,B 0,C 180,E1 -5145.14,E2 -5145.14} C_VEL
LIN {X 0,Y 517.055,Z 195.36,A -85,B 0,C 180,E1 -5145.367,E2 -5145.367} C_VEL
LIN {X 0,Y 517.039,Z 193.045,A -85,B 0,C 180,E1 -5145.775,E2 -5145.775} C_VEL
LIN {X 0,Y 517.369,Z 178.654,A -85,B 0,C 180,E1 -5148.616,E2 -5148.616} C_VEL
LIN {X 0,Y 517.701,Z 164.014,A -85,B 0,C 180,E1 -5151.502,E2 -5151.502} C_VEL
LIN {X 0,Y 518.157,Z 150.076,A -85,B 0,C 180,E1 -5154.331,E2 -5154.331} C_VEL
LIN {X 0,Y 517.656,Z 145.445,A -85,B 0,C 180,E1 -5155.319,E2 -5155.319} C_VEL
LIN {X 0,Y 516.963,Z 141.613,A -85,B 0,C 180,E1 -5156.219,E2 -5156.219} C_VEL
LIN {X 0,Y 516.912,Z 141.596,A -85,B 0,C 180,E1 -5159.523,E2 -5159.523} C_VEL
LIN {X 0,Y 516.897,Z 141.595,A -85,B 0,C 180,E1 -5162.543,E2 -5162.543} C_VEL
LIN {X 0,Y 516.867,Z 141.599,A -85,B 0,C 180,E1 -5165.329,E2 -5165.329} C_VEL
LIN {X 0,Y 516.882,Z 141.601,A -85,B 0,C 180,E1 -5167.943,E2 -5167.943} C_VEL
LIN {X 0,Y 516.883,Z 141.588,A -85,B 0,C 180,E1 -5170.741,E2 -5170.741} C_VEL
LIN {X 0,Y 516.882,Z 141.596,A -85,B 0,C 180,E1 -5172.831,E2 -5172.831} C_VEL
LIN {X 0,Y 516.895,Z 141.595,A -85,B 0,C 180,E1 -5175.006,E2 -5175.006} C_VEL
LIN {X 0,Y 516.912,Z 141.592,A -85,B 0,C 180,E1 -5178.398,E2 -5178.398} C_VEL
LIN {X 0,Y 516.879,Z 141.6,A -85,B 0,C 180,E1 -5181.284,E2 -5181.284} C_VEL
LIN {X 0,Y 516.871,Z 141.595,A -85,B 0,C 180,E1 -5184.219,E2 -5184.219} C_VEL
LIN {X 0,Y 516.895,Z 141.594,A -85,B 0,C 180,E1 -5187.053,E2 -5187.053} C_VEL
LIN {X 0,Y 516.891,Z 141.595,A -85,B 0,C 180,E1 -5189.796,E2 -5189.796} C_VEL
LIN {X 0,Y 516.924,Z 141.586,A -85,B 0,C 180,E1 -5192.467,E2 -5192.467} C_VEL
LIN {X 0,Y 516.907,Z 141.597,A -85,B 0,C 180,E1 -5195.071,E2 -5195.071} C_VEL
LIN {X 0,Y 516.883,Z 141.597,A -85,B 0,C 180,E1 -5198.462,E2 -5198.462} C_VEL
LIN {X 0,Y 516.902,Z 141.59,A -85,B 0,C 180,E1 -5200.954,E2 -5200.954} C_VEL
LIN {X 0,Y 516.911,Z 141.59,A -85,B 0,C 180,E1 -5203.41,E2 -5203.41} C_VEL
LIN {X 0,Y 516.893,Z 141.593,A -85,B 0,C 180,E1 -5205.833,E2 -5205.833} C_VEL
LIN {X 0,Y 516.962,Z 141.585,A -85,B 0,C 180,E1 -5208.233,E2 -5208.233} C_VEL
LIN {X 0,Y 516.965,Z 141.579,A -85,B 0,C 180,E1 -5211.399,E2 -5211.399} C_VEL
LIN {X 0,Y 517.007,Z 141.579,A -85,B 0,C 180,E1 -5213.756,E2 -5213.756} C_VEL
LIN {X 0,Y 517.08,Z 141.569,A -85,B 0,C 180,E1 -5217.663,E2 -5217.663} C_VEL
LIN {X 0,Y 517.09,Z 141.565,A -85,B 0,C 180,E1 -5220.778,E2 -5220.778} C_VEL
LIN {X 0,Y 517.01,Z 141.578,A -85,B 0,C 180,E1 -5223.117,E2 -5223.117} C_VEL
LIN {X 0,Y 517.006,Z 141.586,A -85,B 0,C 180,E1 -5226.243,E2 -5226.243} C_VEL
LIN {X 0,Y 516.949,Z 141.579,A -85,B 0,C 180,E1 -5229.389,E2 -5229.389} C_VEL
LIN {X 0,Y 516.947,Z 141.586,A -85,B 0,C 180,E1 -5231.807,E2 -5231.807} C_VEL
LIN {X 0,Y 516.939,Z 141.588,A -85,B 0,C 180,E1 -5235.146,E2 -5235.146} C_VEL
LIN {X 0,Y 516.921,Z 141.585,A -85,B 0,C 180,E1 -5238.222,E2 -5238.222} C_VEL
LIN {X 0,Y 516.907,Z 141.589,A -85,B 0,C 180,E1 -5240.701,E2 -5240.701} C_VEL
LIN {X 0,Y 516.906,Z 141.596,A -85,B 0,C 180,E1 -5244.072,E2 -5244.072} C_VEL
LIN {X 0,Y 516.924,Z 141.584,A -85,B 0,C 180,E1 -5246.657,E2 -5246.657} C_VEL
LIN {X 0,Y 516.906,Z 141.597,A -85,B 0,C 180,E1 -5249.524,E2 -5249.524} C_VEL
LIN {X 0,Y 516.896,Z 141.593,A -85,B 0,C 180,E1 -5252.544,E2 -5252.544} C_VEL
LIN {X 0,Y 516.879,Z 141.596,A -85,B 0,C 180,E1 -5255.332,E2 -5255.332} C_VEL
LIN {X 0,Y 516.876,Z 141.598,A -85,B 0,C 180,E1 -5257.943,E2 -5257.943} C_VEL
LIN {X 0,Y 516.881,Z 141.593,A -85,B 0,C 180,E1 -5260.741,E2 -5260.741} C_VEL
LIN {X 0,Y 516.9,Z 141.596,A -85,B 0,C 180,E1 -5262.829,E2 -5262.829} C_VEL
LIN {X 0,Y 516.917,Z 141.597,A -85,B 0,C 180,E1 -5265.01,E2 -5265.01} C_VEL
LIN {X 0,Y 516.912,Z 141.577,A -85,B 0,C 180,E1 -5268.398,E2 -5268.398} C_VEL
LIN {X 0,Y 516.877,Z 141.593,A -85,B 0,C 180,E1 -5270.294,E2 -5270.294} C_VEL
LIN {X 0,Y 516.208,Z 141.685,A -85,B 0,C 180,E1 -5270.944,E2 -5270.944} C_VEL
LIN {X 0,Y 513.363,Z 142.036,A -85,B 0,C 180,E1 -5271.999,E2 -5271.999} C_VEL
LIN {X 0,Y 510.956,Z 142.341,A -85,B 0,C 180,E1 -5272.85,E2 -5272.85} C_VEL
LIN {X 0,Y 509.916,Z 142.463,A -85,B 0,C 180,E1 -5273.506,E2 -5273.506} C_VEL
LIN {X 0,Y 509.827,Z 142.471,A -85,B 0,C 180,E1 -5273.729,E2 -5273.729} C_VEL
LIN {X 0,Y 509.858,Z 142.467,A -85,B 0,C 180,E1 -5276.539,E2 -5276.539} C_VEL
LIN {X 0,Y 509.847,Z 142.471,A -85,B 0,C 180,E1 -5279.335,E2 -5279.335} C_VEL
LIN {X 0,Y 509.89,Z 142.466,A -85,B 0,C 180,E1 -5282.055,E2 -5282.055} C_VEL
LIN {X 0,Y 509.873,Z 142.477,A -85,B 0,C 180,E1 -5284.704,E2 -5284.704} C_VEL
LIN {X 0,Y 509.833,Z 142.475,A -85,B 0,C 180,E1 -5287.455,E2 -5287.455} C_VEL
LIN {X 0,Y 509.913,Z 142.466,A -85,B 0,C 180,E1 -5289.845,E2 -5289.845} C_VEL
LIN {X 0,Y 509.881,Z 142.47,A -85,B 0,C 180,E1 -5293.175,E2 -5293.175} C_VEL
LIN {X 0,Y 509.861,Z 142.473,A -85,B 0,C 180,E1 -5295.634,E2 -5295.634} C_VEL
LIN {X 0,Y 509.91,Z 142.468,A -85,B 0,C 180,E1 -5298.875,E2 -5298.875} C_VEL
LIN {X 0,Y 509.949,Z 142.467,A -85,B 0,C 180,E1 -5302.078,E2 -5302.078} C_VEL
LIN {X 0,Y 509.98,Z 142.462,A -85,B 0,C 180,E1 -5304.464,E2 -5304.464} C_VEL
LIN {X 0,Y 510.053,Z 142.452,A -85,B 0,C 180,E1 -5307.631,E2 -5307.631} C_VEL
LIN {X 0,Y 510.061,Z 142.448,A -85,B 0,C 180,E1 -5310.789,E2 -5310.789} C_VEL
LIN {X 0,Y 509.953,Z 142.462,A -85,B 0,C 180,E1 -5313.16,E2 -5313.16} C_VEL
LIN {X 0,Y 509.977,Z 142.46,A -85,B 0,C 180,E1 -5316.33,E2 -5316.33} C_VEL
LIN {X 0,Y 509.913,Z 142.466,A -85,B 0,C 180,E1 -5318.72,E2 -5318.72} C_VEL
LIN {X 0,Y 509.901,Z 142.472,A -85,B 0,C 180,E1 -5321.932,E2 -5321.932} C_VEL
LIN {X 0,Y 509.89,Z 142.473,A -85,B 0,C 180,E1 -5325.242,E2 -5325.242} C_VEL
LIN {X 0,Y 509.885,Z 142.472,A -85,B 0,C 180,E1 -5328.001,E2 -5328.001} C_VEL
LIN {X 0,Y 509.847,Z 142.477,A -85,B 0,C 180,E1 -5331.002,E2 -5331.002} C_VEL
LIN {X 0,Y 509.833,Z 142.481,A -85,B 0,C 180,E1 -5333.563,E2 -5333.563} C_VEL
LIN {X 0,Y 509.908,Z 142.466,A -85,B 0,C 180,E1 -5336.379,E2 -5336.379} C_VEL
LIN {X 0,Y 509.882,Z 142.469,A -85,B 0,C 180,E1 -5338.844,E2 -5338.844} C_VEL
LIN {X 0,Y 509.822,Z 142.479,A -85,B 0,C 180,E1 -5341.59,E2 -5341.59} C_VEL
LIN {X 0,Y 509.847,Z 142.466,A -85,B 0,C 180,E1 -5344.413,E2 -5344.413} C_VEL
LIN {X 0,Y 509.814,Z 142.481,A -85,B 0,C 180,E1 -5347.341,E2 -5347.341} C_VEL
LIN {X 0,Y 509.833,Z 142.472,A -85,B 0,C 180,E1 -5350.382,E2 -5350.382} C_VEL
LIN {X 0,Y 509.819,Z 142.47,A -85,B 0,C 180,E1 -5353.062,E2 -5353.062} C_VEL
LIN {X 0,Y 509.826,Z 142.474,A -85,B 0,C 180,E1 -5355.792,E2 -5355.792} C_VEL
LIN {X 0,Y 509.854,Z 142.476,A -85,B 0,C 180,E1 -5358.575,E2 -5358.575} C_VEL
LIN {X 0,Y 509.846,Z 142.472,A -85,B 0,C 180,E1 -5361.786,E2 -5361.786} C_VEL
LIN {X 0,Y 509.842,Z 142.473,A -85,B 0,C 180,E1 -5364.623,E2 -5364.623} C_VEL
LIN {X 0,Y 509.861,Z 142.469,A -85,B 0,C 180,E1 -5367.481,E2 -5367.481} C_VEL
LIN {X 0,Y 509.853,Z 142.478,A -85,B 0,C 180,E1 -5370.274,E2 -5370.274} C_VEL
LIN {X 0,Y 509.883,Z 142.462,A -85,B 0,C 180,E1 -5372.945,E2 -5372.945} C_VEL
LIN {X 0,Y 509.865,Z 142.469,A -85,B 0,C 180,E1 -5375.574,E2 -5375.574} C_VEL
LIN {X 0,Y 509.818,Z 142.482,A -85,B 0,C 180,E1 -5378.149,E2 -5378.149} C_VEL
LIN {X 0,Y 509.86,Z 142.461,A -85,B 0,C 180,E1 -5380.682,E2 -5380.682} C_VEL
LIN {X 0,Y 509.88,Z 142.465,A -85,B 0,C 180,E1 -5383.175,E2 -5383.175} C_VEL
LIN {X 0,Y 509.86,Z 142.474,A -85,B 0,C 180,E1 -5385.634,E2 -5385.634} C_VEL
LIN {X 0,Y 509.909,Z 142.457,A -85,B 0,C 180,E1 -5388.875,E2 -5388.875} C_VEL
LIN {X 0,Y 509.947,Z 142.462,A -85,B 0,C 180,E1 -5392.079,E2 -5392.079} C_VEL
LIN {X 0,Y 509.978,Z 142.456,A -85,B 0,C 180,E1 -5394.465,E2 -5394.465} C_VEL
LIN {X 0,Y 510.05,Z 142.449,A -85,B 0,C 180,E1 -5397.631,E2 -5397.631} C_VEL
LIN {X 0,Y 510.06,Z 142.436,A -85,B 0,C 180,E1 -5400.79,E2 -5400.79} C_VEL
LIN {X 0,Y 509.952,Z 142.46,A -85,B 0,C 180,E1 -5403.161,E2 -5403.161} C_VEL
LIN {X 0,Y 509.975,Z 142.454,A -85,B 0,C 180,E1 -5406.33,E2 -5406.33} C_VEL
LIN {X 0,Y 509.911,Z 142.457,A -85,B 0,C 180,E1 -5408.721,E2 -5408.721} C_VEL
LIN {X 0,Y 509.901,Z 142.463,A -85,B 0,C 180,E1 -5411.932,E2 -5411.932} C_VEL
LIN {X 0,Y 509.891,Z 142.472,A -85,B 0,C 180,E1 -5415.242,E2 -5415.242} C_VEL
LIN {X 0,Y 509.886,Z 142.458,A -85,B 0,C 180,E1 -5418.001,E2 -5418.001} C_VEL
LIN {X 0,Y 509.848,Z 142.474,A -85,B 0,C 180,E1 -5421.002,E2 -5421.002} C_VEL
LIN {X 0,Y 509.862,Z 142.471,A -85,B 0,C 180,E1 -5424.427,E2 -5424.427} C_VEL
LIN {X 0,Y 509.882,Z 142.466,A -85,B 0,C 180,E1 -5427.056,E2 -5427.056} C_VEL
LIN {X 0,Y 509.856,Z 142.47,A -85,B 0,C 180,E1 -5429.752,E2 -5429.752} C_VEL
LIN {X 0,Y 509.873,Z 142.471,A -85,B 0,C 180,E1 -5432.775,E2 -5432.775} C_VEL
LIN {X 0,Y 509.826,Z 142.472,A -85,B 0,C 180,E1 -5435.579,E2 -5435.579} C_VEL
LIN {X 0,Y 509.848,Z 142.477,A -85,B 0,C 180,E1 -5438.339,E2 -5438.339} C_VEL
LIN {X 0,Y 509.854,Z 142.47,A -85,B 0,C 180,E1 -5441.426,E2 -5441.426} C_VEL
LIN {X 0,Y 509.838,Z 142.477,A -85,B 0,C 180,E1 -5444.67,E2 -5444.67} C_VEL
LIN {X 0,Y 509.833,Z 142.474,A -85,B 0,C 180,E1 -5447.511,E2 -5447.511} C_VEL
LIN {X 0,Y 509.848,Z 142.475,A -85,B 0,C 180,E1 -5450.648,E2 -5450.648} C_VEL
LIN {X 0,Y 509.825,Z 142.476,A -85,B 0,C 180,E1 -5453.647,E2 -5453.647} C_VEL
LIN {X 0,Y 509.86,Z 142.473,A -85,B 0,C 180,E1 -5456.54,E2 -5456.54} C_VEL
LIN {X 0,Y 509.847,Z 142.476,A -85,B 0,C 180,E1 -5459.335,E2 -5459.335} C_VEL
LIN {X 0,Y 509.888,Z 142.471,A -85,B 0,C 180,E1 -5462.055,E2 -5462.055} C_VEL
LIN {X 0,Y 509.929,Z 142.508,A -85,B 0,C 180,E1 -5463.619,E2 -5463.619} C_VEL
LIN {X 0,Y 511.177,Z 150.374,A -85,B 0,C 180,E1 -5465.406,E2 -5465.406} C_VEL
LIN {X 0,Y 510.766,Z 163.882,A -85,B 0,C 180,E1 -5468.191,E2 -5468.191} C_VEL
LIN {X 0,Y 510.396,Z 177.434,A -85,B 0,C 180,E1 -5470.912,E2 -5470.912} C_VEL
LIN {X 0,Y 510.071,Z 191.885,A -85,B 0,C 180,E1 -5473.799,E2 -5473.799} C_VEL
LIN {X 0,Y 510.011,Z 194.894,A -85,B 0,C 180,E1 -5474.394,E2 -5474.394} C_VEL
LIN {X 0,Y 510.966,Z 200.788,A -85,B 0,C 180,E1 -5474.544,E2 -5474.544} C_VEL
LIN {X 0,Y 512.197,Z 209.592,A -85,B 0,C 180,E1 -5474.707,E2 -5474.707} C_VEL
LIN {X 0,Y 511.773,Z 299.81,A -85,B 0,C 180,E1 -5475.993,E2 -5475.993} C_VEL
LIN {X 0,Y 511.567,Z 309.705,A -85,B 0,C 180,E1 -5476.216,E2 -5476.216} C_VEL
LIN {X 0,Y 511.376,Z 319.683,A -85,B 0,C 180,E1 -5476.54,E2 -5476.54} C_VEL
LIN {X 0,Y 511.103,Z 330.047,A -85,B 0,C 180,E1 -5476.987,E2 -5476.987} C_VEL
LIN {X 0,Y 510.819,Z 340.008,A -85,B 0,C 180,E1 -5477.536,E2 -5477.536} C_VEL
LIN {X 0,Y 510.589,Z 348.184,A -85,B 0,C 180,E1 -5478.085,E2 -5478.085} C_VEL
LIN {X 0,Y 510.306,Z 356.915,A -85,B 0,C 180,E1 -5478.783,E2 -5478.783} C_VEL
LIN {X 0,Y 510.073,Z 364.312,A -85,B 0,C 180,E1 -5479.481,E2 -5479.481} C_VEL
LIN {X 0,Y 509.901,Z 371.534,A -85,B 0,C 180,E1 -5480.28,E2 -5480.28} C_VEL
LIN {X 0,Y 509.661,Z 377.735,A -85,B 0,C 180,E1 -5481.076,E2 -5481.076} C_VEL
LIN {X 0,Y 509.492,Z 384.272,A -85,B 0,C 180,E1 -5482.071,E2 -5482.071} C_VEL
LIN {X 0,Y 509.334,Z 389.825,A -85,B 0,C 180,E1 -5483.085,E2 -5483.085} C_VEL
